LIN {X -0.020,Y -573.873,Z 1383.296,A 0.000,B 0.000,C 90.000,E1 89.312} C_DIS
LIN {X 0.144,Y -573.679,Z 1383.294,A 0.000,B 0.000,C 90.000,E1 88.854} C_DIS
LIN {X 0.149,Y -575.125,Z 1383.283,A 0.000,B 0.000,C 90.000,E1 86.963} C_DIS
LIN {X 0.133,Y -576.877,Z 1383.273,A 0.000,B 0.000,C 90.000,E1 85.065} C_DIS
LIN {X -0.055,Y -579.570,Z 1383.259,A 0.000,B 0.000,C 90.000,E1 82.648} C_DIS
LIN {X -0.182,Y -581.188,Z 1383.252,A 0.000,B 0.000,C 90.000,E1 81.310} C_DIS
LIN {X 0.204,Y -582.794,Z 1383.244,A 0.000,B 0.000,C 90.000,E1 79.926} C_DIS
LIN {X 0.003,Y -584.002,Z 1383.238,A 0.000,B 0.000,C 90.000,E1 78.870} C_DIS
LIN {X 0.074,Y -585.294,Z 1383.231,A 0.000,B 0.000,C 90.000,E1 77.521} C_DIS
LIN {X 0.163,Y -586.431,Z 1383.223,A 0.000,B 0.000,C 90.000,E1 76.172} C_DIS
LIN {X 0.161,Y -587.247,Z 1383.217,A 0.000,B 0.000,C 90.000,E1 75.102} C_DIS
LIN {X -0.143,Y -588.135,Z 1383.210,A 0.000,B 0.000,C 90.000,E1 73.795} C_DIS
LIN {X -0.346,Y -589.192,Z 1383.200,A 0.000,B 0.000,C 90.000,E1 71.945} C_DIS
LIN {X -0.162,Y -590.287,Z 1383.189,A 0.000,B 0.000,C 90.000,E1 70.061} C_DIS
LIN {X -0.073,Y -591.511,Z 1383.177,A 0.000,B 0.000,C 90.000,E1 67.922} C_DIS
LIN {X -0.049,Y -593.020,Z 1383.166,A 0.000,B 0.000,C 90.000,E1 65.793} C_DIS
LIN {X -0.080,Y -594.374,Z 1383.157,A 0.000,B 0.000,C 90.000,E1 64.204} C_DIS
LIN {X -0.086,Y -595.616,Z 1383.148,A 0.000,B 0.000,C 90.000,E1 62.615} C_DIS
LIN {X 0.354,Y -598.154,Z 1383.132,A 0.000,B 0.000,C 90.000,E1 59.665} C_DIS
LIN {X -0.139,Y -599.857,Z 1383.121,A 0.000,B 0.000,C 90.000,E1 57.867} C_DIS
LIN {X -0.197,Y -601.333,Z 1383.113,A 0.000,B 0.000,C 90.000,E1 56.294} C_DIS
LIN {X 0.366,Y -602.985,Z 1383.103,A 0.000,B 0.000,C 90.000,E1 54.402} C_DIS
LIN {X 0.223,Y -604.383,Z 1383.094,A 0.000,B 0.000,C 90.000,E1 52.844} C_DIS
LIN {X 0.156,Y -605.045,Z 1383.089,A 0.000,B 0.000,C 90.000,E1 52.065} C_DIS
LIN {X -0.005,Y -605.621,Z 1383.085,A 0.000,B 0.000,C 90.000,E1 51.295} C_DIS
LIN {X -0.206,Y -606.465,Z 1383.076,A 0.000,B 0.000,C 90.000,E1 49.747} C_DIS
LIN {X 0.188,Y -607.019,Z 1383.069,A 0.000,B 0.000,C 90.000,E1 48.405} C_DIS
LIN {X -0.066,Y -607.335,Z 1383.060,A 0.000,B 0.000,C 90.000,E1 46.863} C_DIS
LIN {X -0.150,Y -607.368,Z 1383.053,A 0.000,B 0.000,C 90.000,E1 45.567} C_DIS
LIN {X -0.039,Y -607.232,Z 1383.047,A 0.000,B 0.000,C 90.000,E1 44.514} C_DIS
LIN {X 0.065,Y -606.899,Z 1383.042,A 0.000,B 0.000,C 90.000,E1 43.461} C_DIS
LIN {X -0.256,Y -606.457,Z 1383.036,A 0.000,B 0.000,C 90.000,E1 42.447} C_DIS
LIN {X -0.066,Y -605.580,Z 1383.027,A 0.000,B 0.000,C 90.000,E1 40.862} C_DIS
LIN {X -0.152,Y -604.657,Z 1383.020,A 0.000,B 0.000,C 90.000,E1 39.564} C_DIS
LIN {X 0.157,Y -604.020,Z 1383.015,A 0.000,B 0.000,C 90.000,E1 38.749} C_DIS
LIN {X 0.122,Y -602.737,Z 1383.008,A 0.000,B 0.000,C 90.000,E1 37.443} C_DIS
LIN {X 0.061,Y -601.033,Z 1383.001,A 0.000,B 0.000,C 90.000,E1 36.137} C_DIS
LIN {X -0.040,Y -599.758,Z 1382.996,A 0.000,B 0.000,C 90.000,E1 35.358} C_DIS
LIN {X -0.002,Y -598.228,Z 1382.992,A 0.000,B 0.000,C 90.000,E1 34.565} C_DIS
LIN {X 0.101,Y -595.889,Z 1382.986,A 0.000,B 0.000,C 90.000,E1 33.499} C_DIS
LIN {X 0.221,Y -594.656,Z 1382.983,A 0.000,B 0.000,C 90.000,E1 32.959} C_DIS
LIN {X -0.175,Y -591.080,Z 1382.976,A 0.000,B 0.000,C 90.000,E1 31.671} C_DIS
LIN {X -0.086,Y -589.475,Z 1382.973,A 0.000,B 0.000,C 90.000,E1 31.131} C_DIS
LIN {X -0.127,Y -586.543,Z 1382.969,A 0.000,B 0.000,C 90.000,E1 30.335} C_DIS
LIN {X -0.197,Y -583.338,Z 1382.964,A 0.000,B 0.000,C 90.000,E1 29.539} C_DIS
LIN {X -0.169,Y -580.992,Z 1382.961,A 0.000,B 0.000,C 90.000,E1 28.999} C_DIS
LIN {X 0.203,Y -577.244,Z 1382.957,A 0.000,B 0.000,C 90.000,E1 28.153} C_DIS
LIN {X 0.183,Y -572.284,Z 1382.951,A 0.000,B 0.000,C 90.000,E1 27.206} C_DIS
LIN {X -0.143,Y -566.792,Z 1382.946,A 0.000,B 0.000,C 90.000,E1 26.283} C_DIS
LIN {X 0.003,Y -563.478,Z 1382.943,A 0.000,B 0.000,C 90.000,E1 25.720} C_DIS
LIN {X 0.127,Y -559.951,Z 1382.940,A 0.000,B 0.000,C 90.000,E1 25.155} C_DIS
LIN {X -0.278,Y -556.223,Z 1382.937,A 0.000,B 0.000,C 90.000,E1 24.643} C_DIS
LIN {X -0.203,Y -552.304,Z 1382.934,A 0.000,B 0.000,C 90.000,E1 24.079} C_DIS
LIN {X -0.040,Y -549.189,Z 1382.931,A 0.000,B 0.000,C 90.000,E1 23.643} C_DIS
LIN {X -0.017,Y -544.710,Z 1382.928,A 0.000,B 0.000,C 90.000,E1 23.078} C_DIS
LIN {X 0.218,Y -537.735,Z 1382.924,A 0.000,B 0.000,C 90.000,E1 22.206} C_DIS
LIN {X -0.045,Y -532.751,Z 1382.920,A 0.000,B 0.000,C 90.000,E1 21.663} C_DIS
LIN {X -0.050,Y -522.640,Z 1382.914,A 0.000,B 0.000,C 90.000,E1 20.556} C_DIS
LIN {X -0.068,Y -512.091,Z 1382.908,A 0.000,B 0.000,C 90.000,E1 19.450} C_DIS
LIN {X -0.052,Y -502.768,Z 1382.903,A 0.000,B 0.000,C 90.000,E1 18.489} C_DIS
LIN {X -0.109,Y -486.527,Z 1382.894,A 0.000,B 0.000,C 90.000,E1 16.858} C_DIS
LIN {X -0.241,Y -474.100,Z 1382.887,A 0.000,B 0.000,C 90.000,E1 15.607} C_DIS
LIN {X 0.115,Y -463.083,Z 1382.880,A 0.000,B 0.000,C 90.000,E1 14.426} C_DIS
LIN {X 0.044,Y -449.284,Z 1382.872,A 0.000,B 0.000,C 90.000,E1 13.008} C_DIS
LIN {X -0.001,Y -429.820,Z 1382.861,A 0.000,B 0.000,C 90.000,E1 10.894} C_DIS
LIN {X -0.006,Y -413.486,Z 1382.850,A 0.000,B 0.000,C 90.000,E1 8.973} C_DIS
LIN {X -0.053,Y -403.732,Z 1382.843,A 0.000,B 0.000,C 90.000,E1 7.814} C_DIS
LIN {X 0.113,Y -396.786,Z 1382.839,A 0.000,B 0.000,C 90.000,E1 6.947} C_DIS
LIN {X 0.110,Y -392.848,Z 1382.836,A 0.000,B 0.000,C 90.000,E1 6.429} C_DIS
LIN {X -0.156,Y -390.657,Z 1382.834,A 0.000,B 0.000,C 90.000,E1 6.087} C_DIS
LIN {X -0.193,Y -390.686,Z 1382.834,A 0.000,B 0.000,C 90.000,E1 6.087} C_DIS
LIN {X 0.157,Y -393.696,Z 1382.831,A 0.000,B 0.000,C 90.000,E1 5.625} C_DIS
LIN {X 0.158,Y -398.277,Z 1382.829,A 0.000,B 0.000,C 90.000,E1 5.220} C_DIS
LIN {X 0.115,Y -404.369,Z 1382.827,A 0.000,B 0.000,C 90.000,E1 4.759} C_DIS
LIN {X 0.005,Y -410.468,Z 1382.824,A 0.000,B 0.000,C 90.000,E1 4.245} C_DIS
LIN {X 0.154,Y -417.659,Z 1382.820,A 0.000,B 0.000,C 90.000,E1 3.498} C_DIS
LIN {X 0.153,Y -424.246,Z 1382.815,A 0.000,B 0.000,C 90.000,E1 2.694} C_DIS
LIN {X -0.070,Y -431.567,Z 1382.810,A 0.000,B 0.000,C 90.000,E1 1.718} C_DIS
LIN {X 0.135,Y -437.381,Z 1382.805,A 0.000,B 0.000,C 90.000,E1 0.859} C_DIS
LIN {X 0.000,Y -443.207,Z 1382.800,A 0.000,B 0.000,C 90.000,E1 360.000} C_DIS
LIN {X -0.007,Y -448.622,Z 1382.795,A 0.000,B 0.000,C 90.000,E1 359.141} C_DIS
LIN {X -0.072,Y -453.427,Z 1382.791,A 0.000,B 0.000,C 90.000,E1 358.339} C_DIS
LIN {X -0.079,Y -457.872,Z 1382.786,A 0.000,B 0.000,C 90.000,E1 357.535} C_DIS
LIN {X -0.037,Y -461.977,Z 1382.782,A 0.000,B 0.000,C 90.000,E1 356.731} C_DIS
LIN {X -0.089,Y -465.100,Z 1382.778,A 0.000,B 0.000,C 90.000,E1 356.102} C_DIS
LIN {X 0.021,Y -468.608,Z 1382.774,A 0.000,B 0.000,C 90.000,E1 355.298} C_DIS
LIN {X 0.211,Y -471.931,Z 1382.770,A 0.000,B 0.000,C 90.000,E1 354.489} C_DIS
LIN {X -0.082,Y -474.974,Z 1382.765,A 0.000,B 0.000,C 90.000,E1 353.742} C_DIS
LIN {X -0.176,Y -478.364,Z 1382.760,A 0.000,B 0.000,C 90.000,E1 352.818} C_DIS
LIN {X -0.079,Y -480.443,Z 1382.757,A 0.000,B 0.000,C 90.000,E1 352.186} C_DIS
LIN {X 0.100,Y -482.341,Z 1382.753,A 0.000,B 0.000,C 90.000,E1 351.546} C_DIS
LIN {X -0.042,Y -483.121,Z 1382.751,A 0.000,B 0.000,C 90.000,E1 351.254} C_DIS
LIN {X -0.255,Y -483.750,Z 1382.750,A 0.000,B 0.000,C 90.000,E1 350.971} C_DIS
LIN {X 0.085,Y -484.175,Z 1382.748,A 0.000,B 0.000,C 90.000,E1 350.622} C_DIS
LIN {X -0.048,Y -484.309,Z 1382.746,A 0.000,B 0.000,C 90.000,E1 350.330} C_DIS
LIN {X -0.179,Y -483.925,Z 1382.745,A 0.000,B 0.000,C 90.000,E1 350.038} C_DIS
LIN {X 0.037,Y -483.259,Z 1382.744,A 0.000,B 0.000,C 90.000,E1 349.859} C_DIS
LIN {X 0.166,Y -480.581,Z 1382.743,A 0.000,B 0.000,C 90.000,E1 349.690} C_DIS
LIN {X -0.004,Y -439.598,Z 1382.738,A 0.000,B 0.000,C 90.000,E1 348.757} C_DIS
LIN {X 0.119,Y -404.062,Z 1382.732,A 0.000,B 0.000,C 90.000,E1 347.757} C_DIS
LIN {X -0.141,Y -372.252,Z 1382.726,A 0.000,B 0.000,C 90.000,E1 346.756} C_DIS
LIN {X -0.087,Y -359.594,Z 1382.724,A 0.000,B 0.000,C 90.000,E1 346.284} C_DIS
LIN {X -0.114,Y -359.561,Z 1382.724,A 0.000,B 0.000,C 90.000,E1 346.284} C_DIS
LIN {X 0.021,Y -361.837,Z 1382.684,A 0.000,B 0.000,C 90.000,E1 339.082} C_DIS
LIN {X -0.077,Y -362.147,Z 1382.678,A 0.000,B 0.000,C 90.000,E1 337.975} C_DIS
LIN {X -0.130,Y -366.028,Z 1382.642,A 0.000,B 0.000,C 90.000,E1 331.641} C_DIS
LIN {X -0.029,Y -366.575,Z 1382.636,A 0.000,B 0.000,C 90.000,E1 330.511} C_DIS
LIN {X -0.136,Y -371.414,Z 1382.603,A 0.000,B 0.000,C 90.000,E1 324.609} C_DIS
LIN {X 0.155,Y -371.796,Z 1382.601,A 0.000,B 0.000,C 90.000,E1 324.196} C_DIS
LIN {X -0.057,Y -377.421,Z 1382.567,A 0.000,B 0.000,C 90.000,E1 318.000} C_DIS
LIN {X 0.224,Y -378.265,Z 1382.563,A 0.000,B 0.000,C 90.000,E1 317.229} C_DIS
LIN {X -0.034,Y -384.005,Z 1382.530,A 0.000,B 0.000,C 90.000,E1 311.472} C_DIS
LIN {X 0.014,Y -384.924,Z 1382.526,A 0.000,B 0.000,C 90.000,E1 310.744} C_DIS
LIN {X -0.065,Y -390.676,Z 1382.495,A 0.000,B 0.000,C 90.000,E1 305.025} C_DIS
LIN {X 0.002,Y -391.172,Z 1382.493,A 0.000,B 0.000,C 90.000,E1 304.659} C_DIS
LIN {X -0.156,Y -394.014,Z 1382.473,A 0.000,B 0.000,C 90.000,E1 301.131} C_DIS
LIN {X 0.130,Y -396.888,Z 1382.459,A 0.000,B 0.000,C 90.000,E1 298.615} C_DIS
LIN {X -0.093,Y -397.488,Z 1382.453,A 0.000,B 0.000,C 90.000,E1 297.590} C_DIS
LIN {X 0.141,Y -401.629,Z 1382.426,A 0.000,B 0.000,C 90.000,E1 292.642} C_DIS
LIN {X -0.109,Y -404.701,Z 1382.395,A 0.000,B 0.000,C 90.000,E1 287.094} C_DIS
LIN {X 0.075,Y -405.163,Z 1382.376,A 0.000,B 0.000,C 90.000,E1 283.592} C_DIS
LIN {X -0.116,Y -406.127,Z 1382.364,A 0.000,B 0.000,C 90.000,E1 281.535} C_DIS
LIN {X -0.084,Y -405.826,Z 1382.358,A 0.000,B 0.000,C 90.000,E1 280.489} C_DIS
LIN {X -0.024,Y -405.689,Z 1382.333,A 0.000,B 0.000,C 90.000,E1 275.967} C_DIS
LIN {X 0.014,Y -403.467,Z 1382.304,A 0.000,B 0.000,C 90.000,E1 270.745} C_DIS
LIN {X -0.019,Y -403.254,Z 1382.302,A 0.000,B 0.000,C 90.000,E1 270.401} C_DIS
LIN {X 0.160,Y -398.876,Z 1382.271,A 0.000,B 0.000,C 90.000,E1 264.780} C_DIS
LIN {X 0.058,Y -393.350,Z 1382.244,A 0.000,B 0.000,C 90.000,E1 259.859} C_DIS
LIN {X -0.020,Y -392.780,Z 1382.240,A 0.000,B 0.000,C 90.000,E1 259.162} C_DIS
LIN {X 0.058,Y -386.327,Z 1382.214,A 0.000,B 0.000,C 90.000,E1 254.519} C_DIS
LIN {X 0.020,Y -385.221,Z 1382.208,A 0.000,B 0.000,C 90.000,E1 253.449} C_DIS
LIN {X 0.060,Y -384.022,Z 1382.204,A 0.000,B 0.000,C 90.000,E1 252.725} C_DIS
LIN {X -0.111,Y -377.452,Z 1382.180,A 0.000,B 0.000,C 90.000,E1 248.411} C_DIS
LIN {X -0.018,Y -376.179,Z 1382.174,A 0.000,B 0.000,C 90.000,E1 247.305} C_DIS
LIN {X -0.030,Y -368.350,Z 1382.147,A 0.000,B 0.000,C 90.000,E1 242.538} C_DIS
LIN {X 0.014,Y -366.486,Z 1382.139,A 0.000,B 0.000,C 90.000,E1 241.051} C_DIS
LIN {X 0.098,Y -365.950,Z 1382.137,A 0.000,B 0.000,C 90.000,E1 240.667} C_DIS
LIN {X -0.012,Y -359.125,Z 1382.114,A 0.000,B 0.000,C 90.000,E1 236.580} C_DIS
LIN {X -0.017,Y -356.266,Z 1382.102,A 0.000,B 0.000,C 90.000,E1 234.322} C_DIS
LIN {X 0.204,Y -355.749,Z 1382.100,A 0.000,B 0.000,C 90.000,E1 233.909} C_DIS
LIN {X 0.006,Y -348.729,Z 1382.074,A 0.000,B 0.000,C 90.000,E1 229.380} C_DIS
LIN {X 0.080,Y -346.133,Z 1382.062,A 0.000,B 0.000,C 90.000,E1 227.067} C_DIS
LIN {X 0.207,Y -344.385,Z 1382.055,A 0.000,B 0.000,C 90.000,E1 225.891} C_DIS
LIN {X -0.130,Y -338.157,Z 1382.027,A 0.000,B 0.000,C 90.000,E1 220.906} C_DIS
LIN {X -0.002,Y -336.778,Z 1382.019,A 0.000,B 0.000,C 90.000,E1 219.322} C_DIS
LIN {X -0.107,Y -330.820,Z 1381.988,A 0.000,B 0.000,C 90.000,E1 213.833} C_DIS
LIN {X -0.157,Y -329.265,Z 1381.975,A 0.000,B 0.000,C 90.000,E1 211.465} C_DIS
LIN {X -0.025,Y -324.644,Z 1381.942,A 0.000,B 0.000,C 90.000,E1 205.463} C_DIS
LIN {X -0.130,Y -323.816,Z 1381.928,A 0.000,B 0.000,C 90.000,E1 203.078} C_DIS
LIN {X 0.102,Y -321.071,Z 1381.888,A 0.000,B 0.000,C 90.000,E1 195.843} C_DIS
LIN {X 0.085,Y -321.097,Z 1381.888,A 0.000,B 0.000,C 90.000,E1 195.843} C_DIS
LIN {X -0.157,Y -345.481,Z 1381.882,A 0.000,B 0.000,C 90.000,E1 194.773} C_DIS
LIN {X 0.193,Y -372.735,Z 1381.876,A 0.000,B 0.000,C 90.000,E1 193.647} C_DIS
LIN {X -0.083,Y -401.975,Z 1381.871,A 0.000,B 0.000,C 90.000,E1 192.703} C_DIS
LIN {X 0.166,Y -434.993,Z 1381.865,A 0.000,B 0.000,C 90.000,E1 191.715} C_DIS
LIN {X -0.147,Y -438.036,Z 1381.865,A 0.000,B 0.000,C 90.000,E1 191.658} C_DIS
LIN {X -0.077,Y -439.089,Z 1381.864,A 0.000,B 0.000,C 90.000,E1 191.535} C_DIS
LIN {X -0.202,Y -440.356,Z 1381.862,A 0.000,B 0.000,C 90.000,E1 191.243} C_DIS
LIN {X -0.054,Y -440.972,Z 1381.860,A 0.000,B 0.000,C 90.000,E1 190.894} C_DIS
LIN {X 0.100,Y -441.221,Z 1381.859,A 0.000,B 0.000,C 90.000,E1 190.546} C_DIS
LIN {X -0.019,Y -441.141,Z 1381.855,A 0.000,B 0.000,C 90.000,E1 189.905} C_DIS
LIN {X -0.012,Y -440.794,Z 1381.844,A 0.000,B 0.000,C 90.000,E1 187.936} C_DIS
LIN {X -0.171,Y -440.447,Z 1381.835,A 0.000,B 0.000,C 90.000,E1 186.315} C_DIS
LIN {X -0.100,Y -440.032,Z 1381.828,A 0.000,B 0.000,C 90.000,E1 184.992} C_DIS
LIN {X 0.152,Y -439.714,Z 1381.824,A 0.000,B 0.000,C 90.000,E1 184.302} C_DIS
LIN {X -0.038,Y -439.218,Z 1381.820,A 0.000,B 0.000,C 90.000,E1 183.669} C_DIS
LIN {X -0.126,Y -438.097,Z 1381.815,A 0.000,B 0.000,C 90.000,E1 182.694} C_DIS
LIN {X -0.125,Y -436.311,Z 1381.808,A 0.000,B 0.000,C 90.000,E1 181.375} C_DIS
LIN {X 0.076,Y -435.150,Z 1381.804,A 0.000,B 0.000,C 90.000,E1 180.688} C_DIS
LIN {X -0.165,Y -433.828,Z 1381.800,A 0.000,B 0.000,C 90.000,E1 180.057} C_DIS
LIN {X 0.019,Y -432.334,Z 1381.797,A 0.000,B 0.000,C 90.000,E1 179.370} C_DIS
LIN {X 0.189,Y -430.598,Z 1381.793,A 0.000,B 0.000,C 90.000,E1 178.682} C_DIS
LIN {X -0.001,Y -427.494,Z 1381.787,A 0.000,B 0.000,C 90.000,E1 177.707} C_DIS
LIN {X 0.153,Y -424.395,Z 1381.783,A 0.000,B 0.000,C 90.000,E1 176.849} C_DIS
LIN {X -0.132,Y -420.678,Z 1381.778,A 0.000,B 0.000,C 90.000,E1 176.045} C_DIS
LIN {X 0.000,Y -416.285,Z 1381.773,A 0.000,B 0.000,C 90.000,E1 175.179} C_DIS
LIN {X 0.050,Y -410.147,Z 1381.768,A 0.000,B 0.000,C 90.000,E1 174.147} C_DIS
LIN {X 0.140,Y -398.792,Z 1381.758,A 0.000,B 0.000,C 90.000,E1 172.413} C_DIS
LIN {X -0.071,Y -386.807,Z 1381.747,A 0.000,B 0.000,C 90.000,E1 170.500} C_DIS
LIN {X 0.012,Y -379.002,Z 1381.739,A 0.000,B 0.000,C 90.000,E1 169.050} C_DIS
LIN {X -0.094,Y -376.326,Z 1381.736,A 0.000,B 0.000,C 90.000,E1 168.522} C_DIS
LIN {X -0.041,Y -374.329,Z 1381.733,A 0.000,B 0.000,C 90.000,E1 167.993} C_DIS
LIN {X 0.172,Y -373.011,Z 1381.731,A 0.000,B 0.000,C 90.000,E1 167.521} C_DIS
LIN {X 0.135,Y -373.003,Z 1381.731,A 0.000,B 0.000,C 90.000,E1 167.521} C_DIS
LIN {X 0.176,Y -373.367,Z 1381.729,A 0.000,B 0.000,C 90.000,E1 167.229} C_DIS
LIN {X -0.114,Y -373.475,Z 1381.728,A 0.000,B 0.000,C 90.000,E1 166.992} C_DIS
LIN {X -0.151,Y -373.500,Z 1381.728,A 0.000,B 0.000,C 90.000,E1 166.992} C_DIS
LIN {X 0.019,Y -375.985,Z 1381.725,A 0.000,B 0.000,C 90.000,E1 166.520} C_DIS
LIN {X 0.092,Y -380.278,Z 1381.722,A 0.000,B 0.000,C 90.000,E1 165.936} C_DIS
LIN {X -0.059,Y -387.164,Z 1381.718,A 0.000,B 0.000,C 90.000,E1 165.172} C_DIS
LIN {X 0.124,Y -399.186,Z 1381.711,A 0.000,B 0.000,C 90.000,E1 163.921} C_DIS
LIN {X 0.126,Y -416.360,Z 1381.702,A 0.000,B 0.000,C 90.000,E1 162.362} C_DIS
LIN {X -0.141,Y -440.127,Z 1381.692,A 0.000,B 0.000,C 90.000,E1 160.477} C_DIS
LIN {X -0.186,Y -452.554,Z 1381.686,A 0.000,B 0.000,C 90.000,E1 159.518} C_DIS
LIN {X -0.109,Y -461.794,Z 1381.682,A 0.000,B 0.000,C 90.000,E1 158.773} C_DIS
LIN {X -0.214,Y -467.844,Z 1381.679,A 0.000,B 0.000,C 90.000,E1 158.284} C_DIS
LIN {X 0.106,Y -475.197,Z 1381.676,A 0.000,B 0.000,C 90.000,E1 157.614} C_DIS
LIN {X -0.085,Y -483.917,Z 1381.671,A 0.000,B 0.000,C 90.000,E1 156.847} C_DIS
LIN {X 0.146,Y -493.943,Z 1381.666,A 0.000,B 0.000,C 90.000,E1 155.869} C_DIS
LIN {X -0.013,Y -502.075,Z 1381.661,A 0.000,B 0.000,C 90.000,E1 155.049} C_DIS
LIN {X 0.106,Y -505.969,Z 1381.659,A 0.000,B 0.000,C 90.000,E1 154.613} C_DIS
LIN {X -0.218,Y -513.623,Z 1381.654,A 0.000,B 0.000,C 90.000,E1 153.768} C_DIS
LIN {X 0.072,Y -519.639,Z 1381.650,A 0.000,B 0.000,C 90.000,E1 152.999} C_DIS
LIN {X 0.037,Y -523.026,Z 1381.648,A 0.000,B 0.000,C 90.000,E1 152.564} C_DIS
LIN {X 0.105,Y -527.199,Z 1381.644,A 0.000,B 0.000,C 90.000,E1 151.975} C_DIS
LIN {X 0.206,Y -530.879,Z 1381.641,A 0.000,B 0.000,C 90.000,E1 151.385} C_DIS
LIN {X -0.129,Y -534.105,Z 1381.638,A 0.000,B 0.000,C 90.000,E1 150.845} C_DIS
LIN {X 0.026,Y -536.888,Z 1381.635,A 0.000,B 0.000,C 90.000,E1 150.255} C_DIS
LIN {X -0.073,Y -540.427,Z 1381.630,A 0.000,B 0.000,C 90.000,E1 149.410} C_DIS
LIN {X 0.121,Y -542.498,Z 1381.627,A 0.000,B 0.000,C 90.000,E1 148.820} C_DIS
LIN {X 0.149,Y -544.391,Z 1381.624,A 0.000,B 0.000,C 90.000,E1 148.250} C_DIS
LIN {X 0.109,Y -546.661,Z 1381.619,A 0.000,B 0.000,C 90.000,E1 147.406} C_DIS
LIN {X 0.180,Y -548.004,Z 1381.616,A 0.000,B 0.000,C 90.000,E1 146.834} C_DIS
LIN {X 0.011,Y -549.716,Z 1381.611,A 0.000,B 0.000,C 90.000,E1 146.008} C_DIS
LIN {X -0.196,Y -550.735,Z 1381.608,A 0.000,B 0.000,C 90.000,E1 145.468} C_DIS
LIN {X 0.037,Y -552.308,Z 1381.602,A 0.000,B 0.000,C 90.000,E1 144.322} C_DIS
LIN {X -0.160,Y -552.962,Z 1381.599,A 0.000,B 0.000,C 90.000,E1 143.783} C_DIS
LIN {X 0.108,Y -553.981,Z 1381.593,A 0.000,B 0.000,C 90.000,E1 142.637} C_DIS
LIN {X 0.095,Y -555.227,Z 1381.583,A 0.000,B 0.000,C 90.000,E1 140.964} C_DIS
LIN {X -0.039,Y -556.124,Z 1381.576,A 0.000,B 0.000,C 90.000,E1 139.585} C_DIS
LIN {X -0.074,Y -556.991,Z 1381.566,A 0.000,B 0.000,C 90.000,E1 137.919} C_DIS
LIN {X -0.175,Y -557.566,Z 1381.558,A 0.000,B 0.000,C 90.000,E1 136.539} C_DIS
LIN {X 0.163,Y -558.196,Z 1381.549,A 0.000,B 0.000,C 90.000,E1 134.838} C_DIS
LIN {X 0.061,Y -558.713,Z 1381.542,A 0.000,B 0.000,C 90.000,E1 133.461} C_DIS
LIN {X -0.011,Y -559.084,Z 1381.534,A 0.000,B 0.000,C 90.000,E1 132.081} C_DIS
LIN {X -0.070,Y -559.395,Z 1381.526,A 0.000,B 0.000,C 90.000,E1 130.701} C_DIS
LIN {X -0.123,Y -560.425,Z 1381.511,A 0.000,B 0.000,C 90.000,E1 127.935} C_DIS
LIN {X 0.065,Y -561.015,Z 1381.508,A 0.000,B 0.000,C 90.000,E1 127.363} C_DIS
LIN {X 0.160,Y -561.930,Z 1381.506,A 0.000,B 0.000,C 90.000,E1 127.076} C_DIS
LIN {X 0.173,Y -562.481,Z 1381.505,A 0.000,B 0.000,C 90.000,E1 126.790} C_DIS
LIN {X 0.131,Y -562.526,Z 1381.505,A 0.000,B 0.000,C 90.000,E1 126.790} C_DIS
LIN {X 0.028,Y -563.550,Z 1381.504,A 0.000,B 0.000,C 90.000,E1 126.710} C_DIS
LIN {X 0.110,Y -569.997,Z 1381.503,A 0.000,B 0.000,C 90.000,E1 126.457} C_DIS
LIN {X -0.098,Y -579.785,Z 1381.501,A 0.000,B 0.000,C 90.000,E1 126.217} C_DIS
LIN {X 0.251,Y -582.362,Z 1381.501,A 0.000,B 0.000,C 90.000,E1 126.091} C_DIS
LIN {X -0.258,Y -588.367,Z 1381.499,A 0.000,B 0.000,C 90.000,E1 125.884} C_DIS
LIN {X -0.073,Y -591.151,Z 1381.499,A 0.000,B 0.000,C 90.000,E1 125.724} C_DIS
LIN {X 0.346,Y -594.060,Z 1381.498,A 0.000,B 0.000,C 90.000,E1 125.518} C_DIS
LIN {X -0.120,Y -599.752,Z 1381.495,A 0.000,B 0.000,C 90.000,E1 125.185} C_DIS
LIN {X -0.077,Y -604.019,Z 1381.494,A 0.000,B 0.000,C 90.000,E1 124.865} C_DIS
LIN {X 0.058,Y -609.454,Z 1381.491,A 0.000,B 0.000,C 90.000,E1 124.405} C_DIS
LIN {X -0.097,Y -617.243,Z 1381.487,A 0.000,B 0.000,C 90.000,E1 123.706} C_DIS
LIN {X -0.097,Y -622.157,Z 1381.484,A 0.000,B 0.000,C 90.000,E1 123.214} C_DIS
LIN {X 0.227,Y -627.868,Z 1381.481,A 0.000,B 0.000,C 90.000,E1 122.546} C_DIS
LIN {X -0.297,Y -631.133,Z 1381.479,A 0.000,B 0.000,C 90.000,E1 122.212} C_DIS
LIN {X -0.417,Y -637.998,Z 1381.474,A 0.000,B 0.000,C 90.000,E1 121.337} C_DIS
LIN {X 0.034,Y -642.421,Z 1381.470,A 0.000,B 0.000,C 90.000,E1 120.669} C_DIS
LIN {X -0.035,Y -646.297,Z 1381.467,A 0.000,B 0.000,C 90.000,E1 120.050} C_DIS
LIN {X 0.166,Y -649.593,Z 1381.464,A 0.000,B 0.000,C 90.000,E1 119.411} C_DIS
LIN {X -0.171,Y -652.380,Z 1381.460,A 0.000,B 0.000,C 90.000,E1 118.821} C_DIS
LIN {X 0.033,Y -654.061,Z 1381.457,A 0.000,B 0.000,C 90.000,E1 118.309} C_DIS
LIN {X -0.327,Y -655.509,Z 1381.455,A 0.000,B 0.000,C 90.000,E1 117.847} C_DIS
LIN {X 0.020,Y -656.508,Z 1381.450,A 0.000,B 0.000,C 90.000,E1 117.078} C_DIS
LIN {X 0.139,Y -656.689,Z 1381.449,A 0.000,B 0.000,C 90.000,E1 116.821} C_DIS
LIN {X -0.090,Y -656.521,Z 1381.445,A 0.000,B 0.000,C 90.000,E1 116.104} C_DIS
LIN {X 0.148,Y -656.182,Z 1381.442,A 0.000,B 0.000,C 90.000,E1 115.591} C_DIS
LIN {X 0.265,Y -655.954,Z 1381.441,A 0.000,B 0.000,C 90.000,E1 115.335} C_DIS
LIN {X -0.375,Y -655.110,Z 1381.438,A 0.000,B 0.000,C 90.000,E1 114.899} C_DIS
LIN {X -0.261,Y -654.591,Z 1381.437,A 0.000,B 0.000,C 90.000,E1 114.643} C_DIS
LIN {X 0.012,Y -651.678,Z 1381.433,A 0.000,B 0.000,C 90.000,E1 114.003} C_DIS
LIN {X -0.056,Y -647.230,Z 1381.431,A 0.000,B 0.000,C 90.000,E1 113.515} C_DIS
LIN {X -0.011,Y -645.868,Z 1381.430,A 0.000,B 0.000,C 90.000,E1 113.387} C_DIS
LIN {X -0.021,Y -641.544,Z 1381.429,A 0.000,B 0.000,C 90.000,E1 113.153} C_DIS
LIN {X 0.184,Y -636.673,Z 1381.427,A 0.000,B 0.000,C 90.000,E1 112.898} C_DIS
LIN {X 0.131,Y -631.213,Z 1381.426,A 0.000,B 0.000,C 90.000,E1 112.717} C_DIS
LIN {X 0.064,Y -617.234,Z 1381.424,A 0.000,B 0.000,C 90.000,E1 112.333} C_DIS
LIN {X 0.001,Y -617.209,Z 1381.424,A 0.000,B 0.000,C 90.000,E1 112.333} C_DIS
LIN {X -0.151,Y -623.404,Z 1381.421,A 0.000,B 0.000,C 90.000,E1 111.716} C_DIS
LIN {X 0.198,Y -627.890,Z 1381.418,A 0.000,B 0.000,C 90.000,E1 111.227} C_DIS
LIN {X 0.039,Y -631.423,Z 1381.416,A 0.000,B 0.000,C 90.000,E1 110.865} C_DIS
LIN {X -0.133,Y -636.709,Z 1381.412,A 0.000,B 0.000,C 90.000,E1 110.248} C_DIS
LIN {X -0.238,Y -641.308,Z 1381.409,A 0.000,B 0.000,C 90.000,E1 109.631} C_DIS
LIN {X 0.083,Y -646.030,Z 1381.405,A 0.000,B 0.000,C 90.000,E1 108.852} C_DIS
LIN {X -0.123,Y -650.949,Z 1381.400,A 0.000,B 0.000,C 90.000,E1 108.000} C_DIS
LIN {X 0.339,Y -655.241,Z 1381.395,A 0.000,B 0.000,C 90.000,E1 107.094} C_DIS
LIN {X -0.012,Y -658.153,Z 1381.391,A 0.000,B 0.000,C 90.000,E1 106.386} C_DIS
LIN {X -0.046,Y -659.626,Z 1381.388,A 0.000,B 0.000,C 90.000,E1 105.898} C_DIS
LIN {X -0.353,Y -661.325,Z 1381.384,A 0.000,B 0.000,C 90.000,E1 105.190} C_DIS
LIN {X 0.002,Y -662.557,Z 1381.380,A 0.000,B 0.000,C 90.000,E1 104.426} C_DIS
LIN {X -0.021,Y -663.206,Z 1381.377,A 0.000,B 0.000,C 90.000,E1 103.939} C_DIS
LIN {X -0.203,Y -663.683,Z 1381.375,A 0.000,B 0.000,C 90.000,E1 103.467} C_DIS
LIN {X 0.028,Y -663.975,Z 1381.371,A 0.000,B 0.000,C 90.000,E1 102.715} C_DIS
LIN {X -0.147,Y -663.951,Z 1381.368,A 0.000,B 0.000,C 90.000,E1 102.243} C_DIS
LIN {X -0.324,Y -663.729,Z 1381.365,A 0.000,B 0.000,C 90.000,E1 101.771} C_DIS
LIN {X 0.053,Y -662.928,Z 1381.361,A 0.000,B 0.000,C 90.000,E1 101.007} C_DIS
LIN {X -0.260,Y -662.226,Z 1381.359,A 0.000,B 0.000,C 90.000,E1 100.546} C_DIS
LIN {X 0.195,Y -661.236,Z 1381.356,A 0.000,B 0.000,C 90.000,E1 100.018} C_DIS
LIN {X -0.122,Y -660.068,Z 1381.353,A 0.000,B 0.000,C 90.000,E1 99.557} C_DIS
LIN {X 0.098,Y -657.885,Z 1381.349,A 0.000,B 0.000,C 90.000,E1 98.803} C_DIS
LIN {X -0.232,Y -656.211,Z 1381.346,A 0.000,B 0.000,C 90.000,E1 98.341} C_DIS
LIN {X 0.168,Y -654.322,Z 1381.344,A 0.000,B 0.000,C 90.000,E1 97.814} C_DIS
LIN {X -0.184,Y -652.193,Z 1381.341,A 0.000,B 0.000,C 90.000,E1 97.352} C_DIS
LIN {X -0.126,Y -648.582,Z 1381.337,A 0.000,B 0.000,C 90.000,E1 96.606} C_DIS
LIN {X 0.131,Y -645.841,Z 1381.334,A 0.000,B 0.000,C 90.000,E1 96.087} C_DIS
LIN {X 0.246,Y -642.240,Z 1381.330,A 0.000,B 0.000,C 90.000,E1 95.454} C_DIS
LIN {X 0.134,Y -636.874,Z 1381.326,A 0.000,B 0.000,C 90.000,E1 94.588} C_DIS
LIN {X 0.168,Y -632.492,Z 1381.322,A 0.000,B 0.000,C 90.000,E1 93.955} C_DIS
LIN {X -0.261,Y -628.532,Z 1381.319,A 0.000,B 0.000,C 90.000,E1 93.498} C_DIS
LIN {X -0.294,Y -622.636,Z 1381.316,A 0.000,B 0.000,C 90.000,E1 92.865} C_DIS
LIN {X -0.153,Y -616.126,Z 1381.312,A 0.000,B 0.000,C 90.000,E1 92.236} C_DIS
LIN {X 0.268,Y -609.623,Z 1381.309,A 0.000,B 0.000,C 90.000,E1 91.604} C_DIS
LIN {X 0.112,Y -604.109,Z 1381.307,A 0.000,B 0.000,C 90.000,E1 91.146} C_DIS
LIN {X 0.183,Y -599.489,Z 1381.305,A 0.000,B 0.000,C 90.000,E1 90.802} C_DIS
LIN {X -0.181,Y -596.399,Z 1381.303,A 0.000,B 0.000,C 90.000,E1 90.630} C_DIS
LIN {X -0.172,Y -591.380,Z 1381.302,A 0.000,B 0.000,C 90.000,E1 90.344} C_DIS
LIN {X -0.235,Y -587.734,Z 1381.301,A 0.000,B 0.000,C 90.000,E1 90.172} C_DIS
LIN {X -0.225,Y -582.641,Z 1381.300,A 0.000,B 0.000,C 90.000,E1 89.943} C_DIS
LIN {X -0.128,Y -578.416,Z 1381.298,A 0.000,B 0.000,C 90.000,E1 89.714} C_DIS
LIN {X 0.178,Y -577.051,Z 1381.298,A 0.000,B 0.000,C 90.000,E1 89.599} C_DIS
LIN {X -0.083,Y -574.787,Z 1381.297,A 0.000,B 0.000,C 90.000,E1 89.427} C_DIS
LIN {X -0.097,Y -573.959,Z 1381.296,A 0.000,B 0.000,C 90.000,E1 89.255} C_DIS
LIN {X 0.026,Y -573.666,Z 1381.294,A 0.000,B 0.000,C 90.000,E1 88.854} C_DIS
LIN {X 0.209,Y -575.282,Z 1381.282,A 0.000,B 0.000,C 90.000,E1 86.674} C_DIS
LIN {X 0.252,Y -576.278,Z 1381.276,A 0.000,B 0.000,C 90.000,E1 85.584} C_DIS
LIN {X 0.271,Y -578.238,Z 1381.265,A 0.000,B 0.000,C 90.000,E1 83.685} C_DIS
LIN {X 0.259,Y -580.168,Z 1381.256,A 0.000,B 0.000,C 90.000,E1 82.064} C_DIS
LIN {X 0.291,Y -582.106,Z 1381.247,A 0.000,B 0.000,C 90.000,E1 80.443} C_DIS
LIN {X 0.214,Y -583.660,Z 1381.240,A 0.000,B 0.000,C 90.000,E1 79.106} C_DIS
LIN {X 0.276,Y -585.003,Z 1381.232,A 0.000,B 0.000,C 90.000,E1 77.757} C_DIS
LIN {X 0.037,Y -586.399,Z 1381.223,A 0.000,B 0.000,C 90.000,E1 76.172} C_DIS
LIN {X 0.282,Y -587.398,Z 1381.216,A 0.000,B 0.000,C 90.000,E1 74.810} C_DIS
LIN {X 0.294,Y -588.103,Z 1381.210,A 0.000,B 0.000,C 90.000,E1 73.740} C_DIS
LIN {X 0.084,Y -589.161,Z 1381.199,A 0.000,B 0.000,C 90.000,E1 71.891} C_DIS
LIN {X -0.292,Y -590.254,Z 1381.189,A 0.000,B 0.000,C 90.000,E1 70.061} C_DIS
LIN {X -0.312,Y -591.636,Z 1381.176,A 0.000,B 0.000,C 90.000,E1 67.667} C_DIS
LIN {X -0.182,Y -592.994,Z 1381.166,A 0.000,B 0.000,C 90.000,E1 65.793} C_DIS
LIN {X -0.213,Y -594.354,Z 1381.157,A 0.000,B 0.000,C 90.000,E1 64.204} C_DIS
LIN {X -0.220,Y -595.558,Z 1381.148,A 0.000,B 0.000,C 90.000,E1 62.615} C_DIS
LIN {X 0.003,Y -597.890,Z 1381.133,A 0.000,B 0.000,C 90.000,E1 59.950} C_DIS
LIN {X -0.190,Y -599.608,Z 1381.123,A 0.000,B 0.000,C 90.000,E1 58.122} C_DIS
LIN {X -0.335,Y -601.344,Z 1381.113,A 0.000,B 0.000,C 90.000,E1 56.294} C_DIS
LIN {X -0.359,Y -603.207,Z 1381.101,A 0.000,B 0.000,C 90.000,E1 54.196} C_DIS
LIN {X -0.244,Y -604.851,Z 1381.091,A 0.000,B 0.000,C 90.000,E1 52.351} C_DIS
LIN {X -0.144,Y -605.627,Z 1381.085,A 0.000,B 0.000,C 90.000,E1 51.295} C_DIS
LIN {X 0.117,Y -606.435,Z 1381.076,A 0.000,B 0.000,C 90.000,E1 49.703} C_DIS
LIN {X 0.047,Y -606.979,Z 1381.069,A 0.000,B 0.000,C 90.000,E1 48.405} C_DIS
LIN {X 0.208,Y -607.334,Z 1381.060,A 0.000,B 0.000,C 90.000,E1 46.824} C_DIS
LIN {X -0.046,Y -607.374,Z 1381.052,A 0.000,B 0.000,C 90.000,E1 45.283} C_DIS
LIN {X -0.368,Y -607.180,Z 1381.046,A 0.000,B 0.000,C 90.000,E1 44.271} C_DIS
LIN {X 0.177,Y -606.801,Z 1381.040,A 0.000,B 0.000,C 90.000,E1 43.176} C_DIS
LIN {X -0.140,Y -606.321,Z 1381.034,A 0.000,B 0.000,C 90.000,E1 42.162} C_DIS
LIN {X 0.190,Y -605.598,Z 1381.027,A 0.000,B 0.000,C 90.000,E1 40.825} C_DIS
LIN {X -0.291,Y -604.682,Z 1381.020,A 0.000,B 0.000,C 90.000,E1 39.564} C_DIS
LIN {X 0.018,Y -604.057,Z 1381.015,A 0.000,B 0.000,C 90.000,E1 38.749} C_DIS
LIN {X -0.271,Y -603.060,Z 1381.010,A 0.000,B 0.000,C 90.000,E1 37.729} C_DIS
LIN {X -0.094,Y -601.791,Z 1381.004,A 0.000,B 0.000,C 90.000,E1 36.664} C_DIS
LIN {X -0.181,Y -600.714,Z 1380.999,A 0.000,B 0.000,C 90.000,E1 35.884} C_DIS
LIN {X -0.277,Y -599.385,Z 1380.995,A 0.000,B 0.000,C 90.000,E1 35.105} C_DIS
LIN {X 0.102,Y -597.791,Z 1380.990,A 0.000,B 0.000,C 90.000,E1 34.278} C_DIS
LIN {X 0.089,Y -594.765,Z 1380.983,A 0.000,B 0.000,C 90.000,E1 32.959} C_DIS
LIN {X -0.303,Y -591.160,Z 1380.976,A 0.000,B 0.000,C 90.000,E1 31.671} C_DIS
LIN {X -0.214,Y -589.577,Z 1380.973,A 0.000,B 0.000,C 90.000,E1 31.131} C_DIS
LIN {X -0.253,Y -586.663,Z 1380.968,A 0.000,B 0.000,C 90.000,E1 30.335} C_DIS
LIN {X -0.321,Y -583.442,Z 1380.964,A 0.000,B 0.000,C 90.000,E1 29.539} C_DIS
LIN {X 0.085,Y -579.873,Z 1380.959,A 0.000,B 0.000,C 90.000,E1 28.693} C_DIS
LIN {X 0.009,Y -576.642,Z 1380.956,A 0.000,B 0.000,C 90.000,E1 28.025} C_DIS
LIN {X -0.015,Y -571.687,Z 1380.950,A 0.000,B 0.000,C 90.000,E1 27.078} C_DIS
LIN {X 0.071,Y -565.331,Z 1380.944,A 0.000,B 0.000,C 90.000,E1 25.976} C_DIS
LIN {X 0.112,Y -560.992,Z 1380.941,A 0.000,B 0.000,C 90.000,E1 25.283} C_DIS
LIN {X 0.117,Y -556.337,Z 1380.937,A 0.000,B 0.000,C 90.000,E1 24.591} C_DIS
LIN {X 0.080,Y -551.401,Z 1380.933,A 0.000,B 0.000,C 90.000,E1 23.898} C_DIS
LIN {X 0.000,Y -546.034,Z 1380.929,A 0.000,B 0.000,C 90.000,E1 23.206} C_DIS
LIN {X 0.098,Y -537.822,Z 1380.923,A 0.000,B 0.000,C 90.000,E1 22.206} C_DIS
LIN {X -0.162,Y -532.883,Z 1380.920,A 0.000,B 0.000,C 90.000,E1 21.663} C_DIS
LIN {X -0.158,Y -522.525,Z 1380.914,A 0.000,B 0.000,C 90.000,E1 20.536} C_DIS
LIN {X 0.019,Y -511.863,Z 1380.908,A 0.000,B 0.000,C 90.000,E1 19.396} C_DIS
LIN {X 0.111,Y -503.666,Z 1380.903,A 0.000,B 0.000,C 90.000,E1 18.544} C_DIS
LIN {X 0.070,Y -491.550,Z 1380.896,A 0.000,B 0.000,C 90.000,E1 17.330} C_DIS
LIN {X -0.127,Y -479.031,Z 1380.889,A 0.000,B 0.000,C 90.000,E1 16.079} C_DIS
LIN {X -0.152,Y -465.028,Z 1380.881,A 0.000,B 0.000,C 90.000,E1 14.647} C_DIS
LIN {X 0.125,Y -455.048,Z 1380.876,A 0.000,B 0.000,C 90.000,E1 13.592} C_DIS
LIN {X 0.231,Y -438.499,Z 1380.866,A 0.000,B 0.000,C 90.000,E1 11.827} C_DIS
LIN {X -0.073,Y -417.757,Z 1380.853,A 0.000,B 0.000,C 90.000,E1 9.500} C_DIS
LIN {X -0.085,Y -408.020,Z 1380.846,A 0.000,B 0.000,C 90.000,E1 8.341} C_DIS
LIN {X -0.159,Y -399.550,Z 1380.841,A 0.000,B 0.000,C 90.000,E1 7.352} C_DIS
LIN {X 0.053,Y -394.836,Z 1380.837,A 0.000,B 0.000,C 90.000,E1 6.720} C_DIS
LIN {X 0.024,Y -392.300,Z 1380.835,A 0.000,B 0.000,C 90.000,E1 6.372} C_DIS
LIN {X -0.120,Y -390.927,Z 1380.834,A 0.000,B 0.000,C 90.000,E1 6.144} C_DIS
LIN {X -0.158,Y -390.915,Z 1380.834,A 0.000,B 0.000,C 90.000,E1 6.144} C_DIS
LIN {X -0.159,Y -393.884,Z 1380.832,A 0.000,B 0.000,C 90.000,E1 5.739} C_DIS
LIN {X -0.162,Y -398.460,Z 1380.830,A 0.000,B 0.000,C 90.000,E1 5.334} C_DIS
LIN {X 0.159,Y -406.100,Z 1380.826,A 0.000,B 0.000,C 90.000,E1 4.702} C_DIS
LIN {X -0.189,Y -410.643,Z 1380.824,A 0.000,B 0.000,C 90.000,E1 4.359} C_DIS
LIN {X 0.076,Y -414.971,Z 1380.822,A 0.000,B 0.000,C 90.000,E1 3.898} C_DIS
LIN {X -0.057,Y -417.917,Z 1380.820,A 0.000,B 0.000,C 90.000,E1 3.612} C_DIS
LIN {X -0.160,Y -421.814,Z 1380.817,A 0.000,B 0.000,C 90.000,E1 3.151} C_DIS
LIN {X -0.022,Y -424.617,Z 1380.816,A 0.000,B 0.000,C 90.000,E1 2.808} C_DIS
LIN {X -0.176,Y -432.045,Z 1380.810,A 0.000,B 0.000,C 90.000,E1 1.833} C_DIS
LIN {X 0.091,Y -437.898,Z 1380.806,A 0.000,B 0.000,C 90.000,E1 0.974} C_DIS
LIN {X 0.000,Y -444.515,Z 1380.800,A 0.000,B 0.000,C 90.000,E1 360.000} C_DIS
LIN {X 0.003,Y -449.941,Z 1380.795,A 0.000,B 0.000,C 90.000,E1 359.141} C_DIS
LIN {X -0.134,Y -453.892,Z 1380.792,A 0.000,B 0.000,C 90.000,E1 358.511} C_DIS
LIN {X -0.135,Y -458.427,Z 1380.787,A 0.000,B 0.000,C 90.000,E1 357.707} C_DIS
LIN {X -0.114,Y -462.594,Z 1380.783,A 0.000,B 0.000,C 90.000,E1 356.906} C_DIS
LIN {X -0.028,Y -466.519,Z 1380.778,A 0.000,B 0.000,C 90.000,E1 356.102} C_DIS
LIN {X -0.100,Y -471.380,Z 1380.772,A 0.000,B 0.000,C 90.000,E1 355.008} C_DIS
LIN {X -0.049,Y -473.980,Z 1380.769,A 0.000,B 0.000,C 90.000,E1 354.375} C_DIS
LIN {X -0.148,Y -477.554,Z 1380.764,A 0.000,B 0.000,C 90.000,E1 353.451} C_DIS
LIN {X -0.209,Y -480.846,Z 1380.758,A 0.000,B 0.000,C 90.000,E1 352.527} C_DIS
LIN {X 0.244,Y -483.729,Z 1380.753,A 0.000,B 0.000,C 90.000,E1 351.546} C_DIS
LIN {X -0.102,Y -485.514,Z 1380.750,A 0.000,B 0.000,C 90.000,E1 350.971} C_DIS
LIN {X 0.121,Y -486.976,Z 1380.746,A 0.000,B 0.000,C 90.000,E1 350.330} C_DIS
LIN {X -0.004,Y -487.355,Z 1380.745,A 0.000,B 0.000,C 90.000,E1 350.038} C_DIS
LIN {X -0.124,Y -487.508,Z 1380.743,A 0.000,B 0.000,C 90.000,E1 349.746} C_DIS
LIN {X 0.236,Y -487.289,Z 1380.741,A 0.000,B 0.000,C 90.000,E1 349.398} C_DIS
LIN {X 0.117,Y -486.097,Z 1380.740,A 0.000,B 0.000,C 90.000,E1 349.106} C_DIS
LIN {X 0.169,Y -484.246,Z 1380.739,A 0.000,B 0.000,C 90.000,E1 348.993} C_DIS
LIN {X -0.106,Y -447.059,Z 1380.734,A 0.000,B 0.000,C 90.000,E1 348.117} C_DIS
LIN {X 0.159,Y -411.609,Z 1380.728,A 0.000,B 0.000,C 90.000,E1 347.061} C_DIS
LIN {X 0.103,Y -379.879,Z 1380.722,A 0.000,B 0.000,C 90.000,E1 345.992} C_DIS
LIN {X -0.052,Y -359.595,Z 1380.718,A 0.000,B 0.000,C 90.000,E1 345.227} C_DIS
LIN {X -0.081,Y -359.531,Z 1380.718,A 0.000,B 0.000,C 90.000,E1 345.227} C_DIS
LIN {X -0.107,Y -361.978,Z 1380.682,A 0.000,B 0.000,C 90.000,E1 338.827} C_DIS
LIN {X 0.001,Y -365.933,Z 1380.643,A 0.000,B 0.000,C 90.000,E1 331.719} C_DIS
LIN {X 0.079,Y -366.221,Z 1380.641,A 0.000,B 0.000,C 90.000,E1 331.335} C_DIS
LIN {X -0.024,Y -371.300,Z 1380.604,A 0.000,B 0.000,C 90.000,E1 324.689} C_DIS
LIN {X -0.035,Y -371.728,Z 1380.602,A 0.000,B 0.000,C 90.000,E1 324.322} C_DIS
LIN {X 0.043,Y -377.298,Z 1380.567,A 0.000,B 0.000,C 90.000,E1 318.081} C_DIS
LIN {X -0.211,Y -378.205,Z 1380.563,A 0.000,B 0.000,C 90.000,E1 317.391} C_DIS
LIN {X 0.061,Y -383.877,Z 1380.531,A 0.000,B 0.000,C 90.000,E1 311.553} C_DIS
LIN {X 0.110,Y -384.854,Z 1380.527,A 0.000,B 0.000,C 90.000,E1 310.825} C_DIS
LIN {X 0.032,Y -390.548,Z 1380.495,A 0.000,B 0.000,C 90.000,E1 305.105} C_DIS
LIN {X 0.099,Y -391.039,Z 1380.493,A 0.000,B 0.000,C 90.000,E1 304.739} C_DIS
LIN {X -0.055,Y -391.402,Z 1380.491,A 0.000,B 0.000,C 90.000,E1 304.405} C_DIS
LIN {X -0.111,Y -396.766,Z 1380.460,A 0.000,B 0.000,C 90.000,E1 298.743} C_DIS
LIN {X 0.107,Y -397.100,Z 1380.458,A 0.000,B 0.000,C 90.000,E1 298.359} C_DIS
LIN {X -0.107,Y -401.554,Z 1380.427,A 0.000,B 0.000,C 90.000,E1 292.770} C_DIS
LIN {X 0.034,Y -404.618,Z 1380.395,A 0.000,B 0.000,C 90.000,E1 287.166} C_DIS
LIN {X 0.137,Y -404.756,Z 1380.394,A 0.000,B 0.000,C 90.000,E1 286.804} C_DIS
LIN {X 0.136,Y -406.073,Z 1380.365,A 0.000,B 0.000,C 90.000,E1 281.591} C_DIS
LIN {X 0.144,Y -406.113,Z 1380.363,A 0.000,B 0.000,C 90.000,E1 281.243} C_DIS
LIN {X 0.179,Y -405.669,Z 1380.334,A 0.000,B 0.000,C 90.000,E1 276.030} C_DIS
LIN {X 0.184,Y -405.558,Z 1380.332,A 0.000,B 0.000,C 90.000,E1 275.682} C_DIS
LIN {X -0.145,Y -403.524,Z 1380.305,A 0.000,B 0.000,C 90.000,E1 270.859} C_DIS
LIN {X -0.178,Y -403.315,Z 1380.303,A 0.000,B 0.000,C 90.000,E1 270.516} C_DIS
LIN {X 0.011,Y -398.972,Z 1380.272,A 0.000,B 0.000,C 90.000,E1 264.894} C_DIS
LIN {X -0.183,Y -393.144,Z 1380.242,A 0.000,B 0.000,C 90.000,E1 259.634} C_DIS
LIN {X -0.151,Y -392.878,Z 1380.240,A 0.000,B 0.000,C 90.000,E1 259.275} C_DIS
LIN {X -0.129,Y -386.042,Z 1380.213,A 0.000,B 0.000,C 90.000,E1 254.283} C_DIS
LIN {X -0.082,Y -385.313,Z 1380.209,A 0.000,B 0.000,C 90.000,E1 253.559} C_DIS
LIN {X -0.060,Y -384.854,Z 1380.207,A 0.000,B 0.000,C 90.000,E1 253.196} C_DIS
LIN {X 0.042,Y -378.033,Z 1380.183,A 0.000,B 0.000,C 90.000,E1 248.847} C_DIS
LIN {X -0.081,Y -376.285,Z 1380.174,A 0.000,B 0.000,C 90.000,E1 247.411} C_DIS
LIN {X -0.102,Y -375.731,Z 1380.172,A 0.000,B 0.000,C 90.000,E1 247.050} C_DIS
LIN {X 0.002,Y -368.994,Z 1380.150,A 0.000,B 0.000,C 90.000,E1 242.999} C_DIS
LIN {X -0.095,Y -366.135,Z 1380.138,A 0.000,B 0.000,C 90.000,E1 240.795} C_DIS
LIN {X -0.189,Y -359.265,Z 1380.115,A 0.000,B 0.000,C 90.000,E1 236.707} C_DIS
LIN {X 0.037,Y -355.926,Z 1380.100,A 0.000,B 0.000,C 90.000,E1 234.036} C_DIS
LIN {X 0.128,Y -348.857,Z 1380.075,A 0.000,B 0.000,C 90.000,E1 229.461} C_DIS
LIN {X -0.032,Y -346.235,Z 1380.062,A 0.000,B 0.000,C 90.000,E1 227.187} C_DIS
LIN {X 0.091,Y -345.765,Z 1380.060,A 0.000,B 0.000,C 90.000,E1 226.782} C_DIS
LIN {X 0.051,Y -339.036,Z 1380.032,A 0.000,B 0.000,C 90.000,E1 221.757} C_DIS
LIN {X -0.082,Y -336.890,Z 1380.019,A 0.000,B 0.000,C 90.000,E1 219.439} C_DIS
LIN {X -0.067,Y -331.223,Z 1379.991,A 0.000,B 0.000,C 90.000,E1 214.326} C_DIS
LIN {X -0.009,Y -329.324,Z 1379.975,A 0.000,B 0.000,C 90.000,E1 211.544} C_DIS
LIN {X 0.012,Y -326.426,Z 1379.958,A 0.000,B 0.000,C 90.000,E1 208.359} C_DIS
LIN {X 0.042,Y -323.850,Z 1379.929,A 0.000,B 0.000,C 90.000,E1 203.153} C_DIS
LIN {X -0.024,Y -321.162,Z 1379.895,A 0.000,B 0.000,C 90.000,E1 197.040} C_DIS
LIN {X -0.042,Y -321.177,Z 1379.895,A 0.000,B 0.000,C 90.000,E1 197.040} C_DIS
LIN {X 0.088,Y -345.048,Z 1379.888,A 0.000,B 0.000,C 90.000,E1 195.843} C_DIS
LIN {X -0.053,Y -372.133,Z 1379.882,A 0.000,B 0.000,C 90.000,E1 194.717} C_DIS
LIN {X 0.059,Y -399.391,Z 1379.876,A 0.000,B 0.000,C 90.000,E1 193.703} C_DIS
LIN {X 0.215,Y -432.283,Z 1379.870,A 0.000,B 0.000,C 90.000,E1 192.647} C_DIS
LIN {X -0.101,Y -439.350,Z 1379.869,A 0.000,B 0.000,C 90.000,E1 192.479} C_DIS
LIN {X 0.011,Y -440.524,Z 1379.869,A 0.000,B 0.000,C 90.000,E1 192.355} C_DIS
LIN {X 0.106,Y -441.857,Z 1379.867,A 0.000,B 0.000,C 90.000,E1 192.063} C_DIS
LIN {X -0.174,Y -442.650,Z 1379.865,A 0.000,B 0.000,C 90.000,E1 191.771} C_DIS
LIN {X -0.014,Y -442.992,Z 1379.864,A 0.000,B 0.000,C 90.000,E1 191.422} C_DIS
LIN {X 0.150,Y -443.131,Z 1379.862,A 0.000,B 0.000,C 90.000,E1 191.074} C_DIS
LIN {X -0.055,Y -442.980,Z 1379.854,A 0.000,B 0.000,C 90.000,E1 189.792} C_DIS
LIN {X 0.061,Y -442.722,Z 1379.844,A 0.000,B 0.000,C 90.000,E1 187.814} C_DIS
LIN {X -0.118,Y -442.454,Z 1379.834,A 0.000,B 0.000,C 90.000,E1 186.201} C_DIS
LIN {X -0.014,Y -442.108,Z 1379.827,A 0.000,B 0.000,C 90.000,E1 184.878} C_DIS
LIN {X -0.183,Y -441.824,Z 1379.823,A 0.000,B 0.000,C 90.000,E1 184.245} C_DIS
LIN {X 0.084,Y -441.378,Z 1379.820,A 0.000,B 0.000,C 90.000,E1 183.555} C_DIS
LIN {X 0.021,Y -440.353,Z 1379.814,A 0.000,B 0.000,C 90.000,E1 182.579} C_DIS
LIN {X 0.057,Y -438.747,Z 1379.807,A 0.000,B 0.000,C 90.000,E1 181.260} C_DIS
LIN {X 0.055,Y -436.410,Z 1379.800,A 0.000,B 0.000,C 90.000,E1 179.943} C_DIS
LIN {X 0.158,Y -435.782,Z 1379.798,A 0.000,B 0.000,C 90.000,E1 179.599} C_DIS
LIN {X 0.016,Y -433.292,Z 1379.792,A 0.000,B 0.000,C 90.000,E1 178.625} C_DIS
LIN {X 0.206,Y -431.400,Z 1379.789,A 0.000,B 0.000,C 90.000,E1 177.936} C_DIS
LIN {X -0.063,Y -429.155,Z 1379.785,A 0.000,B 0.000,C 90.000,E1 177.306} C_DIS
LIN {X 0.065,Y -427.262,Z 1379.782,A 0.000,B 0.000,C 90.000,E1 176.788} C_DIS
LIN {X 0.183,Y -424.548,Z 1379.779,A 0.000,B 0.000,C 90.000,E1 176.102} C_DIS
LIN {X -0.051,Y -419.408,Z 1379.773,A 0.000,B 0.000,C 90.000,E1 175.122} C_DIS
LIN {X 0.035,Y -414.433,Z 1379.768,A 0.000,B 0.000,C 90.000,E1 174.261} C_DIS
LIN {X 0.084,Y -406.423,Z 1379.761,A 0.000,B 0.000,C 90.000,E1 173.053} C_DIS
LIN {X -0.055,Y -390.795,Z 1379.748,A 0.000,B 0.000,C 90.000,E1 170.622} C_DIS
LIN {X -0.147,Y -384.646,Z 1379.742,A 0.000,B 0.000,C 90.000,E1 169.567} C_DIS
LIN {X 0.081,Y -380.790,Z 1379.738,A 0.000,B 0.000,C 90.000,E1 168.814} C_DIS
LIN {X -0.100,Y -377.294,Z 1379.734,A 0.000,B 0.000,C 90.000,E1 168.117} C_DIS
LIN {X 0.087,Y -375.099,Z 1379.730,A 0.000,B 0.000,C 90.000,E1 167.409} C_DIS
LIN {X 0.073,Y -374.653,Z 1379.729,A 0.000,B 0.000,C 90.000,E1 167.229} C_DIS
LIN {X -0.034,Y -374.445,Z 1379.728,A 0.000,B 0.000,C 90.000,E1 166.992} C_DIS
LIN {X -0.058,Y -374.452,Z 1379.728,A 0.000,B 0.000,C 90.000,E1 166.992} C_DIS
LIN {X 0.074,Y -376.035,Z 1379.726,A 0.000,B 0.000,C 90.000,E1 166.589} C_DIS
LIN {X -0.062,Y -381.063,Z 1379.722,A 0.000,B 0.000,C 90.000,E1 165.880} C_DIS
LIN {X 0.021,Y -387.022,Z 1379.718,A 0.000,B 0.000,C 90.000,E1 165.172} C_DIS
LIN {X 0.122,Y -397.793,Z 1379.712,A 0.000,B 0.000,C 90.000,E1 164.047} C_DIS
LIN {X -0.051,Y -416.508,Z 1379.702,A 0.000,B 0.000,C 90.000,E1 162.362} C_DIS
LIN {X -0.039,Y -441.917,Z 1379.691,A 0.000,B 0.000,C 90.000,E1 160.315} C_DIS
LIN {X 0.019,Y -454.425,Z 1379.685,A 0.000,B 0.000,C 90.000,E1 159.337} C_DIS
LIN {X 0.069,Y -463.676,Z 1379.681,A 0.000,B 0.000,C 90.000,E1 158.592} C_DIS
LIN {X -0.020,Y -472.643,Z 1379.677,A 0.000,B 0.000,C 90.000,E1 157.847} C_DIS
LIN {X 0.166,Y -478.536,Z 1379.674,A 0.000,B 0.000,C 90.000,E1 157.305} C_DIS
LIN {X -0.015,Y -484.334,Z 1379.671,A 0.000,B 0.000,C 90.000,E1 156.794} C_DIS
LIN {X -0.025,Y -494.320,Z 1379.666,A 0.000,B 0.000,C 90.000,E1 155.845} C_DIS
LIN {X -0.149,Y -502.414,Z 1379.661,A 0.000,B 0.000,C 90.000,E1 155.025} C_DIS
LIN {X -0.188,Y -507.571,Z 1379.658,A 0.000,B 0.000,C 90.000,E1 154.460} C_DIS
LIN {X -0.069,Y -515.137,Z 1379.653,A 0.000,B 0.000,C 90.000,E1 153.563} C_DIS
LIN {X 0.169,Y -519.914,Z 1379.650,A 0.000,B 0.000,C 90.000,E1 152.948} C_DIS
LIN {X -0.089,Y -523.293,Z 1379.647,A 0.000,B 0.000,C 90.000,E1 152.538} C_DIS
LIN {X -0.104,Y -526.507,Z 1379.645,A 0.000,B 0.000,C 90.000,E1 152.103} C_DIS
LIN {X -0.009,Y -530.250,Z 1379.642,A 0.000,B 0.000,C 90.000,E1 151.513} C_DIS
LIN {X -0.031,Y -534.259,Z 1379.638,A 0.000,B 0.000,C 90.000,E1 150.795} C_DIS
LIN {X 0.123,Y -537.010,Z 1379.635,A 0.000,B 0.000,C 90.000,E1 150.205} C_DIS
LIN {X -0.168,Y -539.426,Z 1379.631,A 0.000,B 0.000,C 90.000,E1 149.665} C_DIS
LIN {X 0.030,Y -542.562,Z 1379.627,A 0.000,B 0.000,C 90.000,E1 148.791} C_DIS
LIN {X 0.241,Y -544.440,Z 1379.624,A 0.000,B 0.000,C 90.000,E1 148.201} C_DIS
LIN {X 0.031,Y -546.662,Z 1379.619,A 0.000,B 0.000,C 90.000,E1 147.375} C_DIS
LIN {X -0.152,Y -548.577,Z 1379.614,A 0.000,B 0.000,C 90.000,E1 146.548} C_DIS
LIN {X 0.141,Y -550.207,Z 1379.609,A 0.000,B 0.000,C 90.000,E1 145.674} C_DIS
LIN {X 0.248,Y -551.096,Z 1379.606,A 0.000,B 0.000,C 90.000,E1 145.102} C_DIS
LIN {X 0.171,Y -552.627,Z 1379.600,A 0.000,B 0.000,C 90.000,E1 143.989} C_DIS
LIN {X -0.272,Y -553.926,Z 1379.592,A 0.000,B 0.000,C 90.000,E1 142.637} C_DIS
LIN {X 0.063,Y -555.125,Z 1379.583,A 0.000,B 0.000,C 90.000,E1 140.928} C_DIS
LIN {X -0.001,Y -555.973,Z 1379.575,A 0.000,B 0.000,C 90.000,E1 139.542} C_DIS
LIN {X -0.049,Y -556.882,Z 1379.566,A 0.000,B 0.000,C 90.000,E1 137.877} C_DIS
LIN {X 0.222,Y -557.465,Z 1379.558,A 0.000,B 0.000,C 90.000,E1 136.458} C_DIS
LIN {X 0.107,Y -557.986,Z 1379.551,A 0.000,B 0.000,C 90.000,E1 135.081} C_DIS
LIN {X 0.070,Y -558.611,Z 1379.541,A 0.000,B 0.000,C 90.000,E1 133.419} C_DIS
LIN {X -0.034,Y -558.982,Z 1379.534,A 0.000,B 0.000,C 90.000,E1 132.043} C_DIS
LIN {X 0.319,Y -559.313,Z 1379.526,A 0.000,B 0.000,C 90.000,E1 130.620} C_DIS
LIN {X 0.078,Y -560.041,Z 1379.515,A 0.000,B 0.000,C 90.000,E1 128.705} C_DIS
LIN {X -0.175,Y -560.473,Z 1379.512,A 0.000,B 0.000,C 90.000,E1 128.177} C_DIS
LIN {X 0.044,Y -560.560,Z 1379.511,A 0.000,B 0.000,C 90.000,E1 128.016} C_DIS
LIN {X -0.277,Y -561.198,Z 1379.510,A 0.000,B 0.000,C 90.000,E1 127.729} C_DIS
LIN {X -0.182,Y -561.549,Z 1379.508,A 0.000,B 0.000,C 90.000,E1 127.443} C_DIS
LIN {X -0.194,Y -562.366,Z 1379.507,A 0.000,B 0.000,C 90.000,E1 127.237} C_DIS
LIN {X -0.084,Y -563.266,Z 1379.506,A 0.000,B 0.000,C 90.000,E1 127.156} C_DIS
LIN {X -0.212,Y -565.115,Z 1379.506,A 0.000,B 0.000,C 90.000,E1 127.076} C_DIS
LIN {X 0.214,Y -567.377,Z 1379.505,A 0.000,B 0.000,C 90.000,E1 126.950} C_DIS
LIN {X -0.144,Y -577.506,Z 1379.504,A 0.000,B 0.000,C 90.000,E1 126.710} C_DIS
LIN {X 0.168,Y -580.700,Z 1379.503,A 0.000,B 0.000,C 90.000,E1 126.583} C_DIS
LIN {X -0.087,Y -583.715,Z 1379.503,A 0.000,B 0.000,C 90.000,E1 126.503} C_DIS
LIN {X -0.035,Y -586.375,Z 1379.502,A 0.000,B 0.000,C 90.000,E1 126.377} C_DIS
LIN {X 0.045,Y -589.389,Z 1379.501,A 0.000,B 0.000,C 90.000,E1 126.217} C_DIS
LIN {X -0.060,Y -595.443,Z 1379.499,A 0.000,B 0.000,C 90.000,E1 125.884} C_DIS
LIN {X -0.294,Y -601.139,Z 1379.497,A 0.000,B 0.000,C 90.000,E1 125.518} C_DIS
LIN {X 0.364,Y -606.614,Z 1379.495,A 0.000,B 0.000,C 90.000,E1 125.025} C_DIS
LIN {X -0.219,Y -610.678,Z 1379.493,A 0.000,B 0.000,C 90.000,E1 124.739} C_DIS
LIN {X 0.068,Y -618.323,Z 1379.489,A 0.000,B 0.000,C 90.000,E1 123.992} C_DIS
LIN {X 0.091,Y -624.390,Z 1379.485,A 0.000,B 0.000,C 90.000,E1 123.372} C_DIS
LIN {X -0.099,Y -631.039,Z 1379.481,A 0.000,B 0.000,C 90.000,E1 122.625} C_DIS
LIN {X -0.247,Y -636.127,Z 1379.478,A 0.000,B 0.000,C 90.000,E1 122.005} C_DIS
LIN {X 0.185,Y -640.798,Z 1379.474,A 0.000,B 0.000,C 90.000,E1 121.337} C_DIS
LIN {X -0.253,Y -644.286,Z 1379.471,A 0.000,B 0.000,C 90.000,E1 120.875} C_DIS
LIN {X 0.256,Y -648.035,Z 1379.468,A 0.000,B 0.000,C 90.000,E1 120.207} C_DIS
LIN {X -0.089,Y -651.304,Z 1379.465,A 0.000,B 0.000,C 90.000,E1 119.617} C_DIS
LIN {X -0.146,Y -653.564,Z 1379.462,A 0.000,B 0.000,C 90.000,E1 119.127} C_DIS
LIN {X -0.045,Y -654.542,Z 1379.460,A 0.000,B 0.000,C 90.000,E1 118.871} C_DIS
LIN {X 0.171,Y -656.206,Z 1379.458,A 0.000,B 0.000,C 90.000,E1 118.359} C_DIS
LIN {X 0.285,Y -656.932,Z 1379.456,A 0.000,B 0.000,C 90.000,E1 118.103} C_DIS
LIN {X -0.058,Y -657.848,Z 1379.454,A 0.000,B 0.000,C 90.000,E1 117.641} C_DIS
LIN {X 0.185,Y -658.536,Z 1379.451,A 0.000,B 0.000,C 90.000,E1 117.129} C_DIS
LIN {X -0.028,Y -658.515,Z 1379.447,A 0.000,B 0.000,C 90.000,E1 116.411} C_DIS
LIN {X -0.067,Y -658.343,Z 1379.444,A 0.000,B 0.000,C 90.000,E1 115.924} C_DIS
LIN {X 0.185,Y -657.874,Z 1379.441,A 0.000,B 0.000,C 90.000,E1 115.412} C_DIS
LIN {X -0.286,Y -657.586,Z 1379.440,A 0.000,B 0.000,C 90.000,E1 115.207} C_DIS
LIN {X -0.044,Y -656.672,Z 1379.437,A 0.000,B 0.000,C 90.000,E1 114.695} C_DIS
LIN {X -0.198,Y -655.839,Z 1379.436,A 0.000,B 0.000,C 90.000,E1 114.463} C_DIS
LIN {X 0.033,Y -653.434,Z 1379.433,A 0.000,B 0.000,C 90.000,E1 113.951} C_DIS
LIN {X 0.087,Y -652.445,Z 1379.432,A 0.000,B 0.000,C 90.000,E1 113.823} C_DIS
LIN {X -0.017,Y -648.943,Z 1379.430,A 0.000,B 0.000,C 90.000,E1 113.462} C_DIS
LIN {X 0.028,Y -647.621,Z 1379.430,A 0.000,B 0.000,C 90.000,E1 113.334} C_DIS
LIN {X 0.075,Y -645.527,Z 1379.429,A 0.000,B 0.000,C 90.000,E1 113.206} C_DIS
LIN {X -0.253,Y -638.628,Z 1379.427,A 0.000,B 0.000,C 90.000,E1 112.898} C_DIS
LIN {X 0.259,Y -632.173,Z 1379.426,A 0.000,B 0.000,C 90.000,E1 112.642} C_DIS
LIN {X -0.235,Y -619.065,Z 1379.424,A 0.000,B 0.000,C 90.000,E1 112.333} C_DIS
LIN {X -0.297,Y -619.071,Z 1379.424,A 0.000,B 0.000,C 90.000,E1 112.333} C_DIS
LIN {X -0.213,Y -626.640,Z 1379.420,A 0.000,B 0.000,C 90.000,E1 111.535} C_DIS
LIN {X 0.060,Y -632.195,Z 1379.416,A 0.000,B 0.000,C 90.000,E1 110.918} C_DIS
LIN {X -0.122,Y -636.490,Z 1379.413,A 0.000,B 0.000,C 90.000,E1 110.429} C_DIS
LIN {X -0.260,Y -641.182,Z 1379.410,A 0.000,B 0.000,C 90.000,E1 109.812} C_DIS
LIN {X 0.058,Y -645.926,Z 1379.406,A 0.000,B 0.000,C 90.000,E1 109.033} C_DIS
LIN {X -0.150,Y -650.780,Z 1379.401,A 0.000,B 0.000,C 90.000,E1 108.181} C_DIS
LIN {X -0.384,Y -653.912,Z 1379.398,A 0.000,B 0.000,C 90.000,E1 107.583} C_DIS
LIN {X 0.190,Y -656.256,Z 1379.395,A 0.000,B 0.000,C 90.000,E1 107.040} C_DIS
LIN {X 0.146,Y -658.242,Z 1379.392,A 0.000,B 0.000,C 90.000,E1 106.551} C_DIS
LIN {X -0.073,Y -659.850,Z 1379.389,A 0.000,B 0.000,C 90.000,E1 106.079} C_DIS
LIN {X -0.177,Y -660.626,Z 1379.388,A 0.000,B 0.000,C 90.000,E1 105.843} C_DIS
LIN {X 0.339,Y -662.314,Z 1379.384,A 0.000,B 0.000,C 90.000,E1 105.064} C_DIS
LIN {X 0.151,Y -663.218,Z 1379.381,A 0.000,B 0.000,C 90.000,E1 104.592} C_DIS
LIN {X -0.120,Y -664.202,Z 1379.377,A 0.000,B 0.000,C 90.000,E1 103.883} C_DIS
LIN {X -0.296,Y -664.682,Z 1379.374,A 0.000,B 0.000,C 90.000,E1 103.411} C_DIS
LIN {X 0.094,Y -664.920,Z 1379.370,A 0.000,B 0.000,C 90.000,E1 102.647} C_DIS
LIN {X -0.079,Y -664.875,Z 1379.368,A 0.000,B 0.000,C 90.000,E1 102.175} C_DIS
LIN {X 0.262,Y -664.657,Z 1379.365,A 0.000,B 0.000,C 90.000,E1 101.658} C_DIS
LIN {X -0.002,Y -663.809,Z 1379.361,A 0.000,B 0.000,C 90.000,E1 100.950} C_DIS
LIN {X -0.308,Y -663.057,Z 1379.358,A 0.000,B 0.000,C 90.000,E1 100.489} C_DIS
LIN {X 0.154,Y -662.078,Z 1379.355,A 0.000,B 0.000,C 90.000,E1 99.962} C_DIS
LIN {X -0.156,Y -660.913,Z 1379.353,A 0.000,B 0.000,C 90.000,E1 99.500} C_DIS
LIN {X 0.073,Y -658.650,Z 1379.349,A 0.000,B 0.000,C 90.000,E1 98.746} C_DIS
LIN {X 0.280,Y -656.014,Z 1379.345,A 0.000,B 0.000,C 90.000,E1 97.992} C_DIS
LIN {X -0.060,Y -653.989,Z 1379.342,A 0.000,B 0.000,C 90.000,E1 97.530} C_DIS
LIN {X -0.191,Y -652.919,Z 1379.340,A 0.000,B 0.000,C 90.000,E1 97.296} C_DIS
LIN {X -0.126,Y -649.234,Z 1379.336,A 0.000,B 0.000,C 90.000,E1 96.549} C_DIS
LIN {X 0.136,Y -646.502,Z 1379.334,A 0.000,B 0.000,C 90.000,E1 96.030} C_DIS
LIN {X 0.078,Y -641.350,Z 1379.329,A 0.000,B 0.000,C 90.000,E1 95.163} C_DIS
LIN {X 0.153,Y -637.409,Z 1379.325,A 0.000,B 0.000,C 90.000,E1 94.531} C_DIS
LIN {X 0.324,Y -633.970,Z 1379.323,A 0.000,B 0.000,C 90.000,E1 94.012} C_DIS
LIN {X -0.203,Y -630.026,Z 1379.320,A 0.000,B 0.000,C 90.000,E1 93.555} C_DIS
LIN {X -0.226,Y -624.326,Z 1379.316,A 0.000,B 0.000,C 90.000,E1 92.922} C_DIS
LIN {X 0.031,Y -616.840,Z 1379.312,A 0.000,B 0.000,C 90.000,E1 92.178} C_DIS
LIN {X 0.257,Y -608.872,Z 1379.308,A 0.000,B 0.000,C 90.000,E1 91.432} C_DIS
LIN {X 0.160,Y -603.251,Z 1379.306,A 0.000,B 0.000,C 90.000,E1 90.974} C_DIS
LIN {X -0.097,Y -597.003,Z 1379.303,A 0.000,B 0.000,C 90.000,E1 90.573} C_DIS
LIN {X 0.254,Y -593.685,Z 1379.302,A 0.000,B 0.000,C 90.000,E1 90.344} C_DIS
LIN {X -0.103,Y -588.509,Z 1379.301,A 0.000,B 0.000,C 90.000,E1 90.115} C_DIS
LIN {X -0.177,Y -583.221,Z 1379.299,A 0.000,B 0.000,C 90.000,E1 89.885} C_DIS
LIN {X -0.156,Y -577.502,Z 1379.298,A 0.000,B 0.000,C 90.000,E1 89.599} C_DIS
LIN {X 0.179,Y -576.406,Z 1379.297,A 0.000,B 0.000,C 90.000,E1 89.484} C_DIS
LIN {X -0.054,Y -574.456,Z 1379.296,A 0.000,B 0.000,C 90.000,E1 89.312} C_DIS
LIN {X -0.131,Y -573.909,Z 1379.296,A 0.000,B 0.000,C 90.000,E1 89.198} C_DIS
LIN {X 0.177,Y -573.669,Z 1379.294,A 0.000,B 0.000,C 90.000,E1 88.854} C_DIS
LIN {X 0.181,Y -574.101,Z 1379.289,A 0.000,B 0.000,C 90.000,E1 88.051} C_DIS
LIN {X 0.256,Y -575.983,Z 1379.277,A 0.000,B 0.000,C 90.000,E1 85.869} C_DIS
LIN {X 0.050,Y -578.470,Z 1379.264,A 0.000,B 0.000,C 90.000,E1 83.451} C_DIS
LIN {X -0.031,Y -580.418,Z 1379.255,A 0.000,B 0.000,C 90.000,E1 81.837} C_DIS
LIN {X 0.092,Y -582.332,Z 1379.246,A 0.000,B 0.000,C 90.000,E1 80.208} C_DIS
LIN {X -0.217,Y -583.575,Z 1379.240,A 0.000,B 0.000,C 90.000,E1 79.162} C_DIS
LIN {X -0.154,Y -584.933,Z 1379.232,A 0.000,B 0.000,C 90.000,E1 77.813} C_DIS
LIN {X 0.177,Y -586.342,Z 1379.223,A 0.000,B 0.000,C 90.000,E1 76.172} C_DIS
LIN {X 0.100,Y -587.529,Z 1379.214,A 0.000,B 0.000,C 90.000,E1 74.574} C_DIS
LIN {X -0.208,Y -588.337,Z 1379.207,A 0.000,B 0.000,C 90.000,E1 73.268} C_DIS
LIN {X 0.085,Y -589.259,Z 1379.198,A 0.000,B 0.000,C 90.000,E1 71.638} C_DIS
LIN {X -0.155,Y -590.208,Z 1379.189,A 0.000,B 0.000,C 90.000,E1 70.061} C_DIS
LIN {X -0.177,Y -591.589,Z 1379.176,A 0.000,B 0.000,C 90.000,E1 67.667} C_DIS
LIN {X -0.047,Y -592.942,Z 1379.166,A 0.000,B 0.000,C 90.000,E1 65.793} C_DIS
LIN {X -0.079,Y -594.302,Z 1379.157,A 0.000,B 0.000,C 90.000,E1 64.204} C_DIS
LIN {X -0.087,Y -595.493,Z 1379.148,A 0.000,B 0.000,C 90.000,E1 62.615} C_DIS
LIN {X 0.135,Y -597.830,Z 1379.133,A 0.000,B 0.000,C 90.000,E1 59.950} C_DIS
LIN {X -0.059,Y -599.552,Z 1379.123,A 0.000,B 0.000,C 90.000,E1 58.122} C_DIS
LIN {X -0.205,Y -601.298,Z 1379.113,A 0.000,B 0.000,C 90.000,E1 56.294} C_DIS
LIN {X -0.230,Y -603.157,Z 1379.101,A 0.000,B 0.000,C 90.000,E1 54.196} C_DIS
LIN {X -0.116,Y -604.819,Z 1379.091,A 0.000,B 0.000,C 90.000,E1 52.351} C_DIS
LIN {X -0.017,Y -605.604,Z 1379.085,A 0.000,B 0.000,C 90.000,E1 51.295} C_DIS
LIN {X -0.018,Y -606.282,Z 1379.078,A 0.000,B 0.000,C 90.000,E1 49.989} C_DIS
LIN {X 0.174,Y -606.955,Z 1379.069,A 0.000,B 0.000,C 90.000,E1 48.405} C_DIS
LIN {X 0.110,Y -607.275,Z 1379.062,A 0.000,B 0.000,C 90.000,E1 47.106} C_DIS
LIN {X 0.023,Y -607.360,Z 1379.055,A 0.000,B 0.000,C 90.000,E1 45.810} C_DIS
LIN {X 0.321,Y -607.378,Z 1379.050,A 0.000,B 0.000,C 90.000,E1 45.000} C_DIS
LIN {X 0.241,Y -607.030,Z 1379.043,A 0.000,B 0.000,C 90.000,E1 43.704} C_DIS
LIN {X -0.269,Y -606.462,Z 1379.036,A 0.000,B 0.000,C 90.000,E1 42.447} C_DIS
LIN {X -0.338,Y -605.789,Z 1379.028,A 0.000,B 0.000,C 90.000,E1 41.148} C_DIS
LIN {X 0.041,Y -604.931,Z 1379.021,A 0.000,B 0.000,C 90.000,E1 39.806} C_DIS
LIN {X 0.146,Y -604.094,Z 1379.015,A 0.000,B 0.000,C 90.000,E1 38.749} C_DIS
LIN {X -0.143,Y -603.117,Z 1379.010,A 0.000,B 0.000,C 90.000,E1 37.729} C_DIS
LIN {X 0.035,Y -601.896,Z 1379.004,A 0.000,B 0.000,C 90.000,E1 36.664} C_DIS
LIN {X -0.051,Y -600.823,Z 1378.999,A 0.000,B 0.000,C 90.000,E1 35.884} C_DIS
LIN {X -0.148,Y -599.502,Z 1378.995,A 0.000,B 0.000,C 90.000,E1 35.105} C_DIS
LIN {X -0.006,Y -598.451,Z 1378.992,A 0.000,B 0.000,C 90.000,E1 34.565} C_DIS
LIN {X -0.002,Y -595.529,Z 1378.985,A 0.000,B 0.000,C 90.000,E1 33.245} C_DIS
LIN {X 0.120,Y -594.210,Z 1378.982,A 0.000,B 0.000,C 90.000,E1 32.704} C_DIS
LIN {X -0.169,Y -591.310,Z 1378.976,A 0.000,B 0.000,C 90.000,E1 31.671} C_DIS
LIN {X -0.079,Y -589.730,Z 1378.973,A 0.000,B 0.000,C 90.000,E1 31.131} C_DIS
LIN {X -0.117,Y -586.862,Z 1378.969,A 0.000,B 0.000,C 90.000,E1 30.335} C_DIS
LIN {X -0.184,Y -583.652,Z 1378.964,A 0.000,B 0.000,C 90.000,E1 29.539} C_DIS
LIN {X -0.154,Y -581.322,Z 1378.961,A 0.000,B 0.000,C 90.000,E1 28.999} C_DIS
LIN {X 0.221,Y -577.581,Z 1378.957,A 0.000,B 0.000,C 90.000,E1 28.153} C_DIS
LIN {X 0.127,Y -571.919,Z 1378.951,A 0.000,B 0.000,C 90.000,E1 27.078} C_DIS
LIN {X 0.303,Y -566.379,Z 1378.945,A 0.000,B 0.000,C 90.000,E1 26.104} C_DIS
LIN {X -0.252,Y -561.263,Z 1378.941,A 0.000,B 0.000,C 90.000,E1 25.335} C_DIS
LIN {X -0.141,Y -557.593,Z 1378.938,A 0.000,B 0.000,C 90.000,E1 24.771} C_DIS
LIN {X -0.155,Y -552.674,Z 1378.934,A 0.000,B 0.000,C 90.000,E1 24.079} C_DIS
LIN {X 0.010,Y -549.592,Z 1378.931,A 0.000,B 0.000,C 90.000,E1 23.643} C_DIS
LIN {X 0.035,Y -545.159,Z 1378.928,A 0.000,B 0.000,C 90.000,E1 23.078} C_DIS
LIN {X -0.140,Y -538.220,Z 1378.924,A 0.000,B 0.000,C 90.000,E1 22.259} C_DIS
LIN {X -0.045,Y -531.994,Z 1378.920,A 0.000,B 0.000,C 90.000,E1 21.535} C_DIS
LIN {X -0.160,Y -521.650,Z 1378.913,A 0.000,B 0.000,C 90.000,E1 20.429} C_DIS
LIN {X -0.093,Y -512.454,Z 1378.908,A 0.000,B 0.000,C 90.000,E1 19.450} C_DIS
LIN {X -0.081,Y -503.090,Z 1378.903,A 0.000,B 0.000,C 90.000,E1 18.489} C_DIS
LIN {X -0.205,Y -492.165,Z 1378.897,A 0.000,B 0.000,C 90.000,E1 17.402} C_DIS
LIN {X 0.005,Y -479.865,Z 1378.890,A 0.000,B 0.000,C 90.000,E1 16.134} C_DIS
LIN {X -0.001,Y -465.986,Z 1378.882,A 0.000,B 0.000,C 90.000,E1 14.717} C_DIS
LIN {X 0.029,Y -454.987,Z 1378.876,A 0.000,B 0.000,C 90.000,E1 13.592} C_DIS
LIN {X 0.027,Y -438.241,Z 1378.866,A 0.000,B 0.000,C 90.000,E1 11.827} C_DIS
LIN {X -0.006,Y -420.220,Z 1378.854,A 0.000,B 0.000,C 90.000,E1 9.792} C_DIS
LIN {X -0.148,Y -409.277,Z 1378.847,A 0.000,B 0.000,C 90.000,E1 8.511} C_DIS
LIN {X 0.139,Y -400.763,Z 1378.842,A 0.000,B 0.000,C 90.000,E1 7.473} C_DIS
LIN {X -0.053,Y -396.657,Z 1378.839,A 0.000,B 0.000,C 90.000,E1 7.004} C_DIS
LIN {X -0.064,Y -392.808,Z 1378.836,A 0.000,B 0.000,C 90.000,E1 6.486} C_DIS
LIN {X 0.107,Y -391.408,Z 1378.835,A 0.000,B 0.000,C 90.000,E1 6.201} C_DIS
LIN {X -0.188,Y -391.210,Z 1378.834,A 0.000,B 0.000,C 90.000,E1 6.201} C_DIS
LIN {X 0.164,Y -391.230,Z 1378.834,A 0.000,B 0.000,C 90.000,E1 6.144} C_DIS
LIN {X -0.148,Y -394.173,Z 1378.832,A 0.000,B 0.000,C 90.000,E1 5.796} C_DIS
LIN {X -0.111,Y -399.422,Z 1378.830,A 0.000,B 0.000,C 90.000,E1 5.334} C_DIS
LIN {X -0.082,Y -406.885,Z 1378.826,A 0.000,B 0.000,C 90.000,E1 4.759} C_DIS
LIN {X 0.066,Y -411.375,Z 1378.824,A 0.000,B 0.000,C 90.000,E1 4.359} C_DIS
LIN {X 0.127,Y -417.150,Z 1378.821,A 0.000,B 0.000,C 90.000,E1 3.784} C_DIS
LIN {X -0.178,Y -424.074,Z 1378.817,A 0.000,B 0.000,C 90.000,E1 3.037} C_DIS
LIN {X -0.081,Y -431.436,Z 1378.811,A 0.000,B 0.000,C 90.000,E1 2.064} C_DIS
LIN {X -0.142,Y -439.726,Z 1378.805,A 0.000,B 0.000,C 90.000,E1 0.917} C_DIS
LIN {X 0.000,Y -445.832,Z 1378.800,A 0.000,B 0.000,C 90.000,E1 360.000} C_DIS
LIN {X 0.013,Y -451.276,Z 1378.795,A 0.000,B 0.000,C 90.000,E1 359.141} C_DIS
LIN {X -0.026,Y -456.156,Z 1378.791,A 0.000,B 0.000,C 90.000,E1 358.339} C_DIS
LIN {X -0.101,Y -459.812,Z 1378.787,A 0.000,B 0.000,C 90.000,E1 357.707} C_DIS
LIN {X 0.066,Y -464.781,Z 1378.782,A 0.000,B 0.000,C 90.000,E1 356.731} C_DIS
LIN {X 0.035,Y -467.903,Z 1378.778,A 0.000,B 0.000,C 90.000,E1 356.102} C_DIS
LIN {X -0.019,Y -472.798,Z 1378.772,A 0.000,B 0.000,C 90.000,E1 355.008} C_DIS
LIN {X 0.045,Y -475.377,Z 1378.769,A 0.000,B 0.000,C 90.000,E1 354.375} C_DIS
LIN {X 0.127,Y -477.795,Z 1378.765,A 0.000,B 0.000,C 90.000,E1 353.742} C_DIS
LIN {X 0.067,Y -481.156,Z 1378.760,A 0.000,B 0.000,C 90.000,E1 352.818} C_DIS
LIN {X 0.186,Y -483.204,Z 1378.757,A 0.000,B 0.000,C 90.000,E1 352.186} C_DIS
LIN {X 0.256,Y -486.003,Z 1378.752,A 0.000,B 0.000,C 90.000,E1 351.254} C_DIS
LIN {X -0.196,Y -488.547,Z 1378.746,A 0.000,B 0.000,C 90.000,E1 350.387} C_DIS
LIN {X 0.053,Y -489.872,Z 1378.743,A 0.000,B 0.000,C 90.000,E1 349.746} C_DIS
LIN {X -0.060,Y -490.316,Z 1378.741,A 0.000,B 0.000,C 90.000,E1 349.454} C_DIS
LIN {X -0.169,Y -490.541,Z 1378.740,A 0.000,B 0.000,C 90.000,E1 349.162} C_DIS
LIN {X 0.204,Y -490.459,Z 1378.738,A 0.000,B 0.000,C 90.000,E1 348.814} C_DIS
LIN {X 0.096,Y -489.732,Z 1378.736,A 0.000,B 0.000,C 90.000,E1 348.522} C_DIS
LIN {X -0.246,Y -488.718,Z 1378.735,A 0.000,B 0.000,C 90.000,E1 348.409} C_DIS
LIN {X 0.160,Y -487.027,Z 1378.735,A 0.000,B 0.000,C 90.000,E1 348.285} C_DIS
LIN {X 0.006,Y -448.346,Z 1378.729,A 0.000,B 0.000,C 90.000,E1 347.297} C_DIS
LIN {X -0.169,Y -416.536,Z 1378.724,A 0.000,B 0.000,C 90.000,E1 346.353} C_DIS
LIN {X 0.011,Y -388.407,Z 1378.719,A 0.000,B 0.000,C 90.000,E1 345.338} C_DIS
LIN {X -0.072,Y -360.448,Z 1378.712,A 0.000,B 0.000,C 90.000,E1 344.212} C_DIS
LIN {X 0.063,Y -359.681,Z 1378.712,A 0.000,B 0.000,C 90.000,E1 344.157} C_DIS
LIN {X 0.032,Y -359.624,Z 1378.712,A 0.000,B 0.000,C 90.000,E1 344.157} C_DIS
LIN {X 0.138,Y -361.981,Z 1378.682,A 0.000,B 0.000,C 90.000,E1 338.773} C_DIS
LIN {X -0.092,Y -365.947,Z 1378.643,A 0.000,B 0.000,C 90.000,E1 331.719} C_DIS
LIN {X 0.162,Y -366.226,Z 1378.641,A 0.000,B 0.000,C 90.000,E1 331.307} C_DIS
LIN {X -0.117,Y -371.317,Z 1378.604,A 0.000,B 0.000,C 90.000,E1 324.689} C_DIS
LIN {X 0.174,Y -371.740,Z 1378.602,A 0.000,B 0.000,C 90.000,E1 324.276} C_DIS
LIN {X -0.038,Y -377.789,Z 1378.565,A 0.000,B 0.000,C 90.000,E1 317.715} C_DIS
LIN {X 0.230,Y -378.214,Z 1378.563,A 0.000,B 0.000,C 90.000,E1 317.310} C_DIS
LIN {X -0.033,Y -383.896,Z 1378.531,A 0.000,B 0.000,C 90.000,E1 311.553} C_DIS
LIN {X 0.015,Y -384.867,Z 1378.527,A 0.000,B 0.000,C 90.000,E1 310.825} C_DIS
LIN {X -0.062,Y -390.566,Z 1378.495,A 0.000,B 0.000,C 90.000,E1 305.105} C_DIS
LIN {X 0.004,Y -391.059,Z 1378.493,A 0.000,B 0.000,C 90.000,E1 304.739} C_DIS
LIN {X -0.150,Y -391.410,Z 1378.491,A 0.000,B 0.000,C 90.000,E1 304.405} C_DIS
LIN {X 0.142,Y -396.783,Z 1378.460,A 0.000,B 0.000,C 90.000,E1 298.693} C_DIS
LIN {X 0.012,Y -397.106,Z 1378.458,A 0.000,B 0.000,C 90.000,E1 298.359} C_DIS
LIN {X -0.203,Y -401.568,Z 1378.426,A 0.000,B 0.000,C 90.000,E1 292.770} C_DIS
LIN {X -0.061,Y -404.631,Z 1378.395,A 0.000,B 0.000,C 90.000,E1 287.166} C_DIS
LIN {X 0.041,Y -404.754,Z 1378.393,A 0.000,B 0.000,C 90.000,E1 286.804} C_DIS
LIN {X 0.039,Y -406.081,Z 1378.365,A 0.000,B 0.000,C 90.000,E1 281.591} C_DIS
LIN {X 0.047,Y -406.107,Z 1378.363,A 0.000,B 0.000,C 90.000,E1 281.243} C_DIS
LIN {X 0.083,Y -405.672,Z 1378.334,A 0.000,B 0.000,C 90.000,E1 276.030} C_DIS
LIN {X 0.092,Y -405.305,Z 1378.330,A 0.000,B 0.000,C 90.000,E1 275.334} C_DIS
LIN {X 0.162,Y -403.516,Z 1378.305,A 0.000,B 0.000,C 90.000,E1 270.802} C_DIS
LIN {X 0.130,Y -403.307,Z 1378.303,A 0.000,B 0.000,C 90.000,E1 270.458} C_DIS
LIN {X -0.085,Y -398.961,Z 1378.272,A 0.000,B 0.000,C 90.000,E1 264.894} C_DIS
LIN {X 0.109,Y -393.133,Z 1378.242,A 0.000,B 0.000,C 90.000,E1 259.577} C_DIS
LIN {X 0.141,Y -392.867,Z 1378.240,A 0.000,B 0.000,C 90.000,E1 259.218} C_DIS
LIN {X -0.118,Y -386.028,Z 1378.213,A 0.000,B 0.000,C 90.000,E1 254.267} C_DIS
LIN {X -0.176,Y -385.299,Z 1378.209,A 0.000,B 0.000,C 90.000,E1 253.559} C_DIS
LIN {X -0.154,Y -384.828,Z 1378.207,A 0.000,B 0.000,C 90.000,E1 253.196} C_DIS
LIN {X -0.050,Y -378.015,Z 1378.182,A 0.000,B 0.000,C 90.000,E1 248.847} C_DIS
LIN {X 0.173,Y -376.270,Z 1378.174,A 0.000,B 0.000,C 90.000,E1 247.358} C_DIS
LIN {X -0.195,Y -375.704,Z 1378.172,A 0.000,B 0.000,C 90.000,E1 247.050} C_DIS
LIN {X -0.091,Y -368.974,Z 1378.150,A 0.000,B 0.000,C 90.000,E1 242.999} C_DIS
LIN {X -0.187,Y -366.110,Z 1378.138,A 0.000,B 0.000,C 90.000,E1 240.795} C_DIS
LIN {X 0.217,Y -359.244,Z 1378.115,A 0.000,B 0.000,C 90.000,E1 236.628} C_DIS
LIN {X -0.054,Y -355.902,Z 1378.100,A 0.000,B 0.000,C 90.000,E1 234.036} C_DIS
LIN {X 0.038,Y -348.837,Z 1378.075,A 0.000,B 0.000,C 90.000,E1 229.461} C_DIS
LIN {X 0.114,Y -346.220,Z 1378.062,A 0.000,B 0.000,C 90.000,E1 227.148} C_DIS
LIN {X 0.000,Y -345.740,Z 1378.060,A 0.000,B 0.000,C 90.000,E1 226.782} C_DIS
LIN {X -0.039,Y -339.020,Z 1378.032,A 0.000,B 0.000,C 90.000,E1 221.757} C_DIS
LIN {X 0.042,Y -336.876,Z 1378.019,A 0.000,B 0.000,C 90.000,E1 219.402} C_DIS
LIN {X -0.156,Y -331.210,Z 1377.991,A 0.000,B 0.000,C 90.000,E1 214.326} C_DIS
LIN {X -0.097,Y -329.315,Z 1377.975,A 0.000,B 0.000,C 90.000,E1 211.544} C_DIS
LIN {X -0.151,Y -324.884,Z 1377.944,A 0.000,B 0.000,C 90.000,E1 205.976} C_DIS
LIN {X 0.081,Y -323.846,Z 1377.929,A 0.000,B 0.000,C 90.000,E1 203.131} C_DIS
LIN {X 0.140,Y -321.390,Z 1377.901,A 0.000,B 0.000,C 90.000,E1 198.181} C_DIS
LIN {X 0.122,Y -321.429,Z 1377.901,A 0.000,B 0.000,C 90.000,E1 198.181} C_DIS
LIN {X 0.027,Y -344.379,Z 1377.894,A 0.000,B 0.000,C 90.000,E1 196.985} C_DIS
LIN {X -0.054,Y -369.525,Z 1377.888,A 0.000,B 0.000,C 90.000,E1 195.843} C_DIS
LIN {X -0.189,Y -398.414,Z 1377.882,A 0.000,B 0.000,C 90.000,E1 194.717} C_DIS
LIN {X -0.087,Y -431.142,Z 1377.875,A 0.000,B 0.000,C 90.000,E1 193.592} C_DIS
LIN {X -0.001,Y -438.439,Z 1377.874,A 0.000,B 0.000,C 90.000,E1 193.355} C_DIS
LIN {X 0.014,Y -441.207,Z 1377.874,A 0.000,B 0.000,C 90.000,E1 193.244} C_DIS
LIN {X -0.103,Y -442.320,Z 1377.873,A 0.000,B 0.000,C 90.000,E1 193.119} C_DIS
LIN {X 0.023,Y -443.068,Z 1377.872,A 0.000,B 0.000,C 90.000,E1 192.939} C_DIS
LIN {X 0.051,Y -443.581,Z 1377.871,A 0.000,B 0.000,C 90.000,E1 192.771} C_DIS
LIN {X -0.220,Y -444.253,Z 1377.869,A 0.000,B 0.000,C 90.000,E1 192.479} C_DIS
LIN {X 0.040,Y -444.633,Z 1377.867,A 0.000,B 0.000,C 90.000,E1 192.119} C_DIS
LIN {X 0.208,Y -444.813,Z 1377.866,A 0.000,B 0.000,C 90.000,E1 191.771} C_DIS
LIN {X -0.148,Y -444.896,Z 1377.860,A 0.000,B 0.000,C 90.000,E1 190.838} C_DIS
LIN {X -0.155,Y -444.786,Z 1377.851,A 0.000,B 0.000,C 90.000,E1 189.208} C_DIS
LIN {X -0.063,Y -444.632,Z 1377.840,A 0.000,B 0.000,C 90.000,E1 187.239} C_DIS
LIN {X -0.202,Y -444.394,Z 1377.831,A 0.000,B 0.000,C 90.000,E1 185.625} C_DIS
LIN {X -0.192,Y -444.197,Z 1377.826,A 0.000,B 0.000,C 90.000,E1 184.645} C_DIS
LIN {X 0.219,Y -443.700,Z 1377.820,A 0.000,B 0.000,C 90.000,E1 183.612} C_DIS
LIN {X 0.184,Y -442.866,Z 1377.815,A 0.000,B 0.000,C 90.000,E1 182.636} C_DIS
LIN {X 0.135,Y -441.718,Z 1377.809,A 0.000,B 0.000,C 90.000,E1 181.661} C_DIS
LIN {X -0.061,Y -440.807,Z 1377.806,A 0.000,B 0.000,C 90.000,E1 181.031} C_DIS
LIN {X -0.143,Y -439.195,Z 1377.800,A 0.000,B 0.000,C 90.000,E1 180.057} C_DIS
LIN {X 0.085,Y -437.987,Z 1377.797,A 0.000,B 0.000,C 90.000,E1 179.370} C_DIS
LIN {X -0.136,Y -436.510,Z 1377.793,A 0.000,B 0.000,C 90.000,E1 178.740} C_DIS
LIN {X 0.177,Y -433.585,Z 1377.787,A 0.000,B 0.000,C 90.000,E1 177.707} C_DIS
LIN {X -0.038,Y -430.839,Z 1377.783,A 0.000,B 0.000,C 90.000,E1 176.906} C_DIS
LIN {X 0.165,Y -427.367,Z 1377.778,A 0.000,B 0.000,C 90.000,E1 176.045} C_DIS
LIN {X -0.116,Y -424.253,Z 1377.775,A 0.000,B 0.000,C 90.000,E1 175.412} C_DIS
LIN {X 0.056,Y -419.639,Z 1377.770,A 0.000,B 0.000,C 90.000,E1 174.546} C_DIS
LIN {X 0.089,Y -416.517,Z 1377.767,A 0.000,B 0.000,C 90.000,E1 174.033} C_DIS
LIN {X 0.187,Y -412.077,Z 1377.763,A 0.000,B 0.000,C 90.000,E1 173.337} C_DIS
LIN {X 0.184,Y -397.157,Z 1377.751,A 0.000,B 0.000,C 90.000,E1 171.084} C_DIS
LIN {X -0.007,Y -386.630,Z 1377.741,A 0.000,B 0.000,C 90.000,E1 169.342} C_DIS
LIN {X -0.142,Y -381.670,Z 1377.736,A 0.000,B 0.000,C 90.000,E1 168.465} C_DIS
LIN {X -0.136,Y -378.519,Z 1377.732,A 0.000,B 0.000,C 90.000,E1 167.757} C_DIS
LIN {X -0.225,Y -377.804,Z 1377.731,A 0.000,B 0.000,C 90.000,E1 167.589} C_DIS
LIN {X 0.136,Y -377.254,Z 1377.730,A 0.000,B 0.000,C 90.000,E1 167.353} C_DIS
LIN {X 0.082,Y -376.378,Z 1377.726,A 0.000,B 0.000,C 90.000,E1 166.700} C_DIS
LIN {X 0.046,Y -376.384,Z 1377.726,A 0.000,B 0.000,C 90.000,E1 166.700} C_DIS
LIN {X 0.134,Y -376.808,Z 1377.725,A 0.000,B 0.000,C 90.000,E1 166.533} C_DIS
LIN {X 0.097,Y -376.823,Z 1377.725,A 0.000,B 0.000,C 90.000,E1 166.533} C_DIS
LIN {X 0.015,Y -381.214,Z 1377.722,A 0.000,B 0.000,C 90.000,E1 165.880} C_DIS
LIN {X 0.059,Y -386.578,Z 1377.718,A 0.000,B 0.000,C 90.000,E1 165.227} C_DIS
LIN {X 0.167,Y -394.198,Z 1377.714,A 0.000,B 0.000,C 90.000,E1 164.393} C_DIS
LIN {X 0.065,Y -403.474,Z 1377.708,A 0.000,B 0.000,C 90.000,E1 163.504} C_DIS
LIN {X 0.052,Y -418.941,Z 1377.701,A 0.000,B 0.000,C 90.000,E1 162.127} C_DIS
LIN {X 0.068,Y -444.174,Z 1377.690,A 0.000,B 0.000,C 90.000,E1 160.115} C_DIS
LIN {X -0.023,Y -456.714,Z 1377.684,A 0.000,B 0.000,C 90.000,E1 159.156} C_DIS
LIN {X -0.020,Y -465.905,Z 1377.680,A 0.000,B 0.000,C 90.000,E1 158.411} C_DIS
LIN {X -0.210,Y -473.420,Z 1377.677,A 0.000,B 0.000,C 90.000,E1 157.794} C_DIS
LIN {X 0.100,Y -480.762,Z 1377.673,A 0.000,B 0.000,C 90.000,E1 157.102} C_DIS
LIN {X 0.040,Y -489.373,Z 1377.668,A 0.000,B 0.000,C 90.000,E1 156.305} C_DIS
LIN {X -0.208,Y -494.990,Z 1377.665,A 0.000,B 0.000,C 90.000,E1 155.793} C_DIS
LIN {X 0.146,Y -501.817,Z 1377.661,A 0.000,B 0.000,C 90.000,E1 155.049} C_DIS
LIN {X -0.196,Y -505.732,Z 1377.659,A 0.000,B 0.000,C 90.000,E1 154.665} C_DIS
LIN {X -0.065,Y -513.396,Z 1377.654,A 0.000,B 0.000,C 90.000,E1 153.768} C_DIS
LIN {X 0.245,Y -519.411,Z 1377.650,A 0.000,B 0.000,C 90.000,E1 152.999} C_DIS
LIN {X 0.047,Y -523.889,Z 1377.647,A 0.000,B 0.000,C 90.000,E1 152.436} C_DIS
LIN {X -0.189,Y -527.034,Z 1377.645,A 0.000,B 0.000,C 90.000,E1 152.025} C_DIS
LIN {X -0.087,Y -530.724,Z 1377.641,A 0.000,B 0.000,C 90.000,E1 151.435} C_DIS
LIN {X 0.043,Y -533.942,Z 1377.638,A 0.000,B 0.000,C 90.000,E1 150.845} C_DIS
LIN {X 0.057,Y -537.337,Z 1377.634,A 0.000,B 0.000,C 90.000,E1 150.127} C_DIS
LIN {X 0.095,Y -540.232,Z 1377.630,A 0.000,B 0.000,C 90.000,E1 149.410} C_DIS
LIN {X -0.176,Y -542.311,Z 1377.627,A 0.000,B 0.000,C 90.000,E1 148.869} C_DIS
LIN {X 0.031,Y -544.172,Z 1377.624,A 0.000,B 0.000,C 90.000,E1 148.280} C_DIS
LIN {X -0.186,Y -546.438,Z 1377.619,A 0.000,B 0.000,C 90.000,E1 147.454} C_DIS
LIN {X 0.084,Y -548.340,Z 1377.614,A 0.000,B 0.000,C 90.000,E1 146.580} C_DIS
LIN {X -0.087,Y -549.960,Z 1377.610,A 0.000,B 0.000,C 90.000,E1 145.754} C_DIS
LIN {X 0.017,Y -550.851,Z 1377.607,A 0.000,B 0.000,C 90.000,E1 145.182} C_DIS
LIN {X -0.067,Y -552.414,Z 1377.600,A 0.000,B 0.000,C 90.000,E1 144.069} C_DIS
LIN {X 0.192,Y -553.492,Z 1377.594,A 0.000,B 0.000,C 90.000,E1 142.924} C_DIS
LIN {X 0.030,Y -554.333,Z 1377.588,A 0.000,B 0.000,C 90.000,E1 141.823} C_DIS
LIN {X -0.046,Y -555.285,Z 1377.580,A 0.000,B 0.000,C 90.000,E1 140.436} C_DIS
LIN {X 0.245,Y -556.089,Z 1377.573,A 0.000,B 0.000,C 90.000,E1 139.013} C_DIS
LIN {X 0.129,Y -556.845,Z 1377.565,A 0.000,B 0.000,C 90.000,E1 137.634} C_DIS
LIN {X -0.001,Y -557.418,Z 1377.557,A 0.000,B 0.000,C 90.000,E1 136.257} C_DIS
LIN {X -0.050,Y -558.024,Z 1377.548,A 0.000,B 0.000,C 90.000,E1 134.595} C_DIS
LIN {X -0.157,Y -558.542,Z 1377.540,A 0.000,B 0.000,C 90.000,E1 133.218} C_DIS
LIN {X -0.233,Y -558.946,Z 1377.532,A 0.000,B 0.000,C 90.000,E1 131.838} C_DIS
LIN {X 0.041,Y -559.239,Z 1377.526,A 0.000,B 0.000,C 90.000,E1 130.701} C_DIS
LIN {X 0.152,Y -560.132,Z 1377.515,A 0.000,B 0.000,C 90.000,E1 128.749} C_DIS
LIN {X -0.230,Y -560.796,Z 1377.512,A 0.000,B 0.000,C 90.000,E1 128.096} C_DIS
LIN {X 0.178,Y -561.155,Z 1377.511,A 0.000,B 0.000,C 90.000,E1 127.890} C_DIS
LIN {X 0.136,Y -561.202,Z 1377.511,A 0.000,B 0.000,C 90.000,E1 127.890} C_DIS
LIN {X -0.135,Y -562.314,Z 1377.510,A 0.000,B 0.000,C 90.000,E1 127.810} C_DIS
LIN {X 0.085,Y -563.333,Z 1377.509,A 0.000,B 0.000,C 90.000,E1 127.649} C_DIS
LIN {X 0.027,Y -563.777,Z 1377.509,A 0.000,B 0.000,C 90.000,E1 127.569} C_DIS
LIN {X 0.187,Y -567.967,Z 1377.508,A 0.000,B 0.000,C 90.000,E1 127.363} C_DIS
LIN {X -0.116,Y -573.871,Z 1377.507,A 0.000,B 0.000,C 90.000,E1 127.237} C_DIS
LIN {X -0.025,Y -580.529,Z 1377.506,A 0.000,B 0.000,C 90.000,E1 127.030} C_DIS
LIN {X -0.155,Y -586.666,Z 1377.504,A 0.000,B 0.000,C 90.000,E1 126.790} C_DIS
LIN {X 0.128,Y -592.423,Z 1377.503,A 0.000,B 0.000,C 90.000,E1 126.457} C_DIS
LIN {X -0.082,Y -596.627,Z 1377.501,A 0.000,B 0.000,C 90.000,E1 126.217} C_DIS
LIN {X 0.049,Y -599.523,Z 1377.500,A 0.000,B 0.000,C 90.000,E1 126.011} C_DIS
LIN {X -0.105,Y -605.107,Z 1377.498,A 0.000,B 0.000,C 90.000,E1 125.598} C_DIS
LIN {X -0.295,Y -607.855,Z 1377.496,A 0.000,B 0.000,C 90.000,E1 125.391} C_DIS
LIN {X -0.159,Y -614.093,Z 1377.493,A 0.000,B 0.000,C 90.000,E1 124.818} C_DIS
LIN {X -0.055,Y -619.105,Z 1377.491,A 0.000,B 0.000,C 90.000,E1 124.326} C_DIS
LIN {X -0.018,Y -623.888,Z 1377.488,A 0.000,B 0.000,C 90.000,E1 123.833} C_DIS
LIN {X 0.324,Y -628.527,Z 1377.485,A 0.000,B 0.000,C 90.000,E1 123.293} C_DIS
LIN {X 0.158,Y -633.926,Z 1377.482,A 0.000,B 0.000,C 90.000,E1 122.673} C_DIS
LIN {X 0.029,Y -638.755,Z 1377.478,A 0.000,B 0.000,C 90.000,E1 122.054} C_DIS
LIN {X 0.121,Y -642.501,Z 1377.475,A 0.000,B 0.000,C 90.000,E1 121.544} C_DIS
LIN {X 0.027,Y -645.846,Z 1377.473,A 0.000,B 0.000,C 90.000,E1 121.052} C_DIS
LIN {X -0.342,Y -649.588,Z 1377.469,A 0.000,B 0.000,C 90.000,E1 120.463} C_DIS
LIN {X 0.163,Y -652.309,Z 1377.466,A 0.000,B 0.000,C 90.000,E1 119.922} C_DIS
LIN {X -0.157,Y -655.093,Z 1377.463,A 0.000,B 0.000,C 90.000,E1 119.333} C_DIS
LIN {X -0.048,Y -656.094,Z 1377.462,A 0.000,B 0.000,C 90.000,E1 119.077} C_DIS
LIN {X -0.280,Y -658.535,Z 1377.458,A 0.000,B 0.000,C 90.000,E1 118.359} C_DIS
LIN {X 0.095,Y -659.986,Z 1377.453,A 0.000,B 0.000,C 90.000,E1 117.590} C_DIS
LIN {X 0.225,Y -660.247,Z 1377.452,A 0.000,B 0.000,C 90.000,E1 117.334} C_DIS
LIN {X -0.099,Y -660.395,Z 1377.449,A 0.000,B 0.000,C 90.000,E1 116.873} C_DIS
LIN {X 0.297,Y -660.252,Z 1377.445,A 0.000,B 0.000,C 90.000,E1 116.104} C_DIS
LIN {X -0.034,Y -659.886,Z 1377.443,A 0.000,B 0.000,C 90.000,E1 115.643} C_DIS
LIN {X -0.059,Y -659.339,Z 1377.440,A 0.000,B 0.000,C 90.000,E1 115.155} C_DIS
LIN {X 0.197,Y -658.386,Z 1377.437,A 0.000,B 0.000,C 90.000,E1 114.643} C_DIS
LIN {X 0.322,Y -657.648,Z 1377.436,A 0.000,B 0.000,C 90.000,E1 114.387} C_DIS
LIN {X -0.307,Y -655.149,Z 1377.433,A 0.000,B 0.000,C 90.000,E1 113.951} C_DIS
LIN {X -0.250,Y -654.268,Z 1377.432,A 0.000,B 0.000,C 90.000,E1 113.823} C_DIS
LIN {X -0.255,Y -649.363,Z 1377.430,A 0.000,B 0.000,C 90.000,E1 113.334} C_DIS
LIN {X -0.164,Y -647.572,Z 1377.429,A 0.000,B 0.000,C 90.000,E1 113.206} C_DIS
LIN {X 0.169,Y -645.650,Z 1377.428,A 0.000,B 0.000,C 90.000,E1 113.078} C_DIS
LIN {X 0.289,Y -640.429,Z 1377.427,A 0.000,B 0.000,C 90.000,E1 112.823} C_DIS
LIN {X 0.001,Y -638.424,Z 1377.427,A 0.000,B 0.000,C 90.000,E1 112.770} C_DIS
LIN {X -0.087,Y -634.208,Z 1377.426,A 0.000,B 0.000,C 90.000,E1 112.642} C_DIS
LIN {X -0.026,Y -620.762,Z 1377.424,A 0.000,B 0.000,C 90.000,E1 112.280} C_DIS
LIN {X -0.090,Y -620.807,Z 1377.424,A 0.000,B 0.000,C 90.000,E1 112.280} C_DIS
LIN {X -0.226,Y -628.650,Z 1377.419,A 0.000,B 0.000,C 90.000,E1 111.461} C_DIS
LIN {X 0.164,Y -633.310,Z 1377.416,A 0.000,B 0.000,C 90.000,E1 110.918} C_DIS
LIN {X -0.010,Y -637.542,Z 1377.414,A 0.000,B 0.000,C 90.000,E1 110.429} C_DIS
LIN {X -0.138,Y -642.128,Z 1377.410,A 0.000,B 0.000,C 90.000,E1 109.812} C_DIS
LIN {X 0.375,Y -646.073,Z 1377.407,A 0.000,B 0.000,C 90.000,E1 109.141} C_DIS
LIN {X -0.040,Y -650.833,Z 1377.402,A 0.000,B 0.000,C 90.000,E1 108.308} C_DIS
LIN {X -0.071,Y -653.984,Z 1377.398,A 0.000,B 0.000,C 90.000,E1 107.692} C_DIS
LIN {X -0.321,Y -656.352,Z 1377.396,A 0.000,B 0.000,C 90.000,E1 107.221} C_DIS
LIN {X 0.269,Y -658.429,Z 1377.393,A 0.000,B 0.000,C 90.000,E1 106.677} C_DIS
LIN {X 0.159,Y -659.414,Z 1377.391,A 0.000,B 0.000,C 90.000,E1 106.441} C_DIS
LIN {X 0.031,Y -661.729,Z 1377.387,A 0.000,B 0.000,C 90.000,E1 105.717} C_DIS
LIN {X -0.256,Y -663.383,Z 1377.383,A 0.000,B 0.000,C 90.000,E1 105.009} C_DIS
LIN {X 0.205,Y -664.287,Z 1377.381,A 0.000,B 0.000,C 90.000,E1 104.481} C_DIS
LIN {X -0.051,Y -665.210,Z 1377.377,A 0.000,B 0.000,C 90.000,E1 103.772} C_DIS
LIN {X -0.218,Y -665.642,Z 1377.374,A 0.000,B 0.000,C 90.000,E1 103.300} C_DIS
LIN {X 0.267,Y -665.842,Z 1377.371,A 0.000,B 0.000,C 90.000,E1 102.771} C_DIS
LIN {X 0.021,Y -665.746,Z 1377.367,A 0.000,B 0.000,C 90.000,E1 102.063} C_DIS
LIN {X -0.147,Y -665.479,Z 1377.364,A 0.000,B 0.000,C 90.000,E1 101.591} C_DIS
LIN {X 0.204,Y -664.963,Z 1377.362,A 0.000,B 0.000,C 90.000,E1 101.074} C_DIS
LIN {X 0.029,Y -664.234,Z 1377.359,A 0.000,B 0.000,C 90.000,E1 100.602} C_DIS
LIN {X 0.288,Y -662.773,Z 1377.355,A 0.000,B 0.000,C 90.000,E1 99.849} C_DIS
LIN {X 0.092,Y -661.573,Z 1377.352,A 0.000,B 0.000,C 90.000,E1 99.378} C_DIS
LIN {X -0.221,Y -660.090,Z 1377.349,A 0.000,B 0.000,C 90.000,E1 98.916} C_DIS
LIN {X -0.003,Y -657.495,Z 1377.345,A 0.000,B 0.000,C 90.000,E1 98.163} C_DIS
LIN {X 0.314,Y -655.561,Z 1377.343,A 0.000,B 0.000,C 90.000,E1 97.644} C_DIS
LIN {X -0.029,Y -653.392,Z 1377.340,A 0.000,B 0.000,C 90.000,E1 97.182} C_DIS
LIN {X 0.117,Y -649.651,Z 1377.336,A 0.000,B 0.000,C 90.000,E1 96.429} C_DIS
LIN {X -0.221,Y -647.625,Z 1377.334,A 0.000,B 0.000,C 90.000,E1 96.087} C_DIS
LIN {X 0.255,Y -641.660,Z 1377.328,A 0.000,B 0.000,C 90.000,E1 95.049} C_DIS
LIN {X -0.179,Y -638.522,Z 1377.325,A 0.000,B 0.000,C 90.000,E1 94.588} C_DIS
LIN {X -0.128,Y -634.123,Z 1377.322,A 0.000,B 0.000,C 90.000,E1 93.955} C_DIS
LIN {X -0.021,Y -630.199,Z 1377.319,A 0.000,B 0.000,C 90.000,E1 93.440} C_DIS
LIN {X -0.045,Y -624.387,Z 1377.316,A 0.000,B 0.000,C 90.000,E1 92.808} C_DIS
LIN {X 0.051,Y -617.985,Z 1377.312,A 0.000,B 0.000,C 90.000,E1 92.178} C_DIS
LIN {X 0.284,Y -610.127,Z 1377.308,A 0.000,B 0.000,C 90.000,E1 91.432} C_DIS
LIN {X 0.137,Y -604.449,Z 1377.306,A 0.000,B 0.000,C 90.000,E1 90.974} C_DIS
LIN {X 0.165,Y -603.039,Z 1377.305,A 0.000,B 0.000,C 90.000,E1 90.859} C_DIS
LIN {X 0.040,Y -596.805,Z 1377.303,A 0.000,B 0.000,C 90.000,E1 90.458} C_DIS
LIN {X -0.165,Y -593.301,Z 1377.302,A 0.000,B 0.000,C 90.000,E1 90.286} C_DIS
LIN {X 0.112,Y -588.172,Z 1377.300,A 0.000,B 0.000,C 90.000,E1 90.000} C_DIS
LIN {X 0.135,Y -578.358,Z 1377.298,A 0.000,B 0.000,C 90.000,E1 89.542} C_DIS
LIN {X -0.092,Y -576.981,Z 1377.297,A 0.000,B 0.000,C 90.000,E1 89.484} C_DIS
LIN {X 0.258,Y -575.962,Z 1377.297,A 0.000,B 0.000,C 90.000,E1 89.370} C_DIS
LIN {X -0.123,Y -574.061,Z 1377.296,A 0.000,B 0.000,C 90.000,E1 89.198} C_DIS
LIN {X 0.105,Y -573.770,Z 1377.295,A 0.000,B 0.000,C 90.000,E1 89.026} C_DIS
LIN {X 0.249,Y -573.630,Z 1377.293,A 0.000,B 0.000,C 90.000,E1 88.740} C_DIS
LIN {X 0.121,Y -574.090,Z 1377.289,A 0.000,B 0.000,C 90.000,E1 87.993} C_DIS
LIN {X 0.195,Y -575.946,Z 1377.277,A 0.000,B 0.000,C 90.000,E1 85.812} C_DIS
LIN {X -0.221,Y -578.167,Z 1377.265,A 0.000,B 0.000,C 90.000,E1 83.685} C_DIS
LIN {X 0.119,Y -579.765,Z 1377.257,A 0.000,B 0.000,C 90.000,E1 82.299} C_DIS
LIN {X -0.091,Y -581.384,Z 1377.250,A 0.000,B 0.000,C 90.000,E1 80.971} C_DIS
LIN {X 0.049,Y -583.290,Z 1377.241,A 0.000,B 0.000,C 90.000,E1 79.342} C_DIS
LIN {X 0.100,Y -584.679,Z 1377.233,A 0.000,B 0.000,C 90.000,E1 77.993} C_DIS
LIN {X -0.147,Y -586.103,Z 1377.224,A 0.000,B 0.000,C 90.000,E1 76.408} C_DIS
LIN {X -0.228,Y -587.301,Z 1377.216,A 0.000,B 0.000,C 90.000,E1 74.810} C_DIS
LIN {X 0.025,Y -588.149,Z 1377.208,A 0.000,B 0.000,C 90.000,E1 73.449} C_DIS
LIN {X 0.313,Y -589.110,Z 1377.199,A 0.000,B 0.000,C 90.000,E1 71.819} C_DIS
LIN {X -0.254,Y -590.175,Z 1377.189,A 0.000,B 0.000,C 90.000,E1 70.007} C_DIS
LIN {X -0.061,Y -591.576,Z 1377.176,A 0.000,B 0.000,C 90.000,E1 67.592} C_DIS
LIN {X 0.178,Y -593.433,Z 1377.162,A 0.000,B 0.000,C 90.000,E1 65.177} C_DIS
LIN {X -0.295,Y -594.492,Z 1377.155,A 0.000,B 0.000,C 90.000,E1 63.896} C_DIS
LIN {X 0.056,Y -595.482,Z 1377.147,A 0.000,B 0.000,C 90.000,E1 62.538} C_DIS
LIN {X 0.376,Y -597.564,Z 1377.134,A 0.000,B 0.000,C 90.000,E1 60.127} C_DIS
LIN {X -0.041,Y -599.059,Z 1377.125,A 0.000,B 0.000,C 90.000,E1 58.584} C_DIS
LIN {X 0.073,Y -600.540,Z 1377.117,A 0.000,B 0.000,C 90.000,E1 56.993} C_DIS
LIN {X -0.129,Y -601.530,Z 1377.111,A 0.000,B 0.000,C 90.000,E1 55.960} C_DIS
LIN {X -0.055,Y -603.171,Z 1377.101,A 0.000,B 0.000,C 90.000,E1 54.116} C_DIS
LIN {X -0.197,Y -604.613,Z 1377.092,A 0.000,B 0.000,C 90.000,E1 52.557} C_DIS
LIN {X -0.213,Y -605.598,Z 1377.085,A 0.000,B 0.000,C 90.000,E1 51.251} C_DIS
LIN {X -0.097,Y -606.142,Z 1377.079,A 0.000,B 0.000,C 90.000,E1 50.194} C_DIS
LIN {X 0.295,Y -606.752,Z 1377.072,A 0.000,B 0.000,C 90.000,E1 48.852} C_DIS
LIN {X -0.024,Y -607.110,Z 1377.066,A 0.000,B 0.000,C 90.000,E1 47.838} C_DIS
LIN {X 0.107,Y -607.317,Z 1377.060,A 0.000,B 0.000,C 90.000,E1 46.782} C_DIS
LIN {X -0.163,Y -607.383,Z 1377.051,A 0.000,B 0.000,C 90.000,E1 45.243} C_DIS
LIN {X -0.241,Y -607.084,Z 1377.044,A 0.000,B 0.000,C 90.000,E1 43.947} C_DIS
LIN {X 0.048,Y -606.799,Z 1377.040,A 0.000,B 0.000,C 90.000,E1 43.137} C_DIS
LIN {X -0.020,Y -606.170,Z 1377.032,A 0.000,B 0.000,C 90.000,E1 41.838} C_DIS
LIN {X 0.106,Y -605.595,Z 1377.027,A 0.000,B 0.000,C 90.000,E1 40.782} C_DIS
LIN {X 0.224,Y -604.912,Z 1377.021,A 0.000,B 0.000,C 90.000,E1 39.725} C_DIS
LIN {X -0.264,Y -603.833,Z 1377.014,A 0.000,B 0.000,C 90.000,E1 38.463} C_DIS
LIN {X 0.291,Y -602.830,Z 1377.008,A 0.000,B 0.000,C 90.000,E1 37.363} C_DIS
LIN {X -0.023,Y -601.580,Z 1377.002,A 0.000,B 0.000,C 90.000,E1 36.343} C_DIS
LIN {X 0.370,Y -600.427,Z 1376.998,A 0.000,B 0.000,C 90.000,E1 35.518} C_DIS
LIN {X 0.264,Y -598.994,Z 1376.993,A 0.000,B 0.000,C 90.000,E1 34.739} C_DIS
LIN {X -0.064,Y -596.115,Z 1376.986,A 0.000,B 0.000,C 90.000,E1 33.452} C_DIS
LIN {X 0.061,Y -594.878,Z 1376.983,A 0.000,B 0.000,C 90.000,E1 32.911} C_DIS
LIN {X -0.111,Y -592.771,Z 1376.979,A 0.000,B 0.000,C 90.000,E1 32.133} C_DIS
LIN {X 0.075,Y -589.614,Z 1376.973,A 0.000,B 0.000,C 90.000,E1 31.052} C_DIS
LIN {X 0.033,Y -586.729,Z 1376.968,A 0.000,B 0.000,C 90.000,E1 30.256} C_DIS
LIN {X -0.040,Y -583.550,Z 1376.964,A 0.000,B 0.000,C 90.000,E1 29.461} C_DIS
LIN {X 0.362,Y -579.967,Z 1376.959,A 0.000,B 0.000,C 90.000,E1 28.615} C_DIS
LIN {X 0.012,Y -576.715,Z 1376.955,A 0.000,B 0.000,C 90.000,E1 27.975} C_DIS
LIN {X 0.254,Y -571.727,Z 1376.950,A 0.000,B 0.000,C 90.000,E1 27.001} C_DIS
LIN {X 0.173,Y -566.165,Z 1376.945,A 0.000,B 0.000,C 90.000,E1 26.052} C_DIS
LIN {X 0.270,Y -560.130,Z 1376.940,A 0.000,B 0.000,C 90.000,E1 25.079} C_DIS
LIN {X -0.035,Y -557.329,Z 1376.937,A 0.000,B 0.000,C 90.000,E1 24.695} C_DIS
LIN {X 0.325,Y -551.341,Z 1376.933,A 0.000,B 0.000,C 90.000,E1 23.823} C_DIS
LIN {X 0.024,Y -545.943,Z 1376.929,A 0.000,B 0.000,C 90.000,E1 23.153} C_DIS
LIN {X -0.106,Y -540.111,Z 1376.925,A 0.000,B 0.000,C 90.000,E1 22.461} C_DIS
LIN {X 0.128,Y -532.884,Z 1376.920,A 0.000,B 0.000,C 90.000,E1 21.589} C_DIS
LIN {X 0.064,Y -522.567,Z 1376.914,A 0.000,B 0.000,C 90.000,E1 20.482} C_DIS
LIN {X 0.125,Y -513.411,Z 1376.908,A 0.000,B 0.000,C 90.000,E1 19.504} C_DIS
LIN {X -0.197,Y -502.387,Z 1376.902,A 0.000,B 0.000,C 90.000,E1 18.417} C_DIS
LIN {X 0.239,Y -491.612,Z 1376.896,A 0.000,B 0.000,C 90.000,E1 17.275} C_DIS
LIN {X 0.122,Y -479.030,Z 1376.889,A 0.000,B 0.000,C 90.000,E1 16.024} C_DIS
LIN {X -0.186,Y -466.397,Z 1376.882,A 0.000,B 0.000,C 90.000,E1 14.773} C_DIS
LIN {X 0.017,Y -455.010,Z 1376.876,A 0.000,B 0.000,C 90.000,E1 13.592} C_DIS
LIN {X 0.035,Y -438.238,Z 1376.866,A 0.000,B 0.000,C 90.000,E1 11.827} C_DIS
LIN {X 0.009,Y -421.596,Z 1376.855,A 0.000,B 0.000,C 90.000,E1 9.962} C_DIS
LIN {X 0.174,Y -410.484,Z 1376.848,A 0.000,B 0.000,C 90.000,E1 8.624} C_DIS
LIN {X -0.145,Y -400.757,Z 1376.842,A 0.000,B 0.000,C 90.000,E1 7.530} C_DIS
LIN {X 0.069,Y -396.614,Z 1376.839,A 0.000,B 0.000,C 90.000,E1 7.004} C_DIS
LIN {X 0.195,Y -392.208,Z 1376.836,A 0.000,B 0.000,C 90.000,E1 6.372} C_DIS
LIN {X -0.163,Y -391.456,Z 1376.835,A 0.000,B 0.000,C 90.000,E1 6.258} C_DIS
LIN {X 0.188,Y -391.449,Z 1376.835,A 0.000,B 0.000,C 90.000,E1 6.201} C_DIS
LIN {X -0.009,Y -394.254,Z 1376.833,A 0.000,B 0.000,C 90.000,E1 5.853} C_DIS
LIN {X -0.004,Y -399.553,Z 1376.830,A 0.000,B 0.000,C 90.000,E1 5.391} C_DIS
LIN {X 0.082,Y -405.455,Z 1376.828,A 0.000,B 0.000,C 90.000,E1 4.935} C_DIS
LIN {X -0.134,Y -410.246,Z 1376.825,A 0.000,B 0.000,C 90.000,E1 4.588} C_DIS
LIN {X -0.158,Y -417.525,Z 1376.822,A 0.000,B 0.000,C 90.000,E1 3.898} C_DIS
LIN {X 0.161,Y -424.353,Z 1376.817,A 0.000,B 0.000,C 90.000,E1 3.094} C_DIS
LIN {X -0.040,Y -430.847,Z 1376.813,A 0.000,B 0.000,C 90.000,E1 2.293} C_DIS
LIN {X 0.222,Y -438.120,Z 1376.807,A 0.000,B 0.000,C 90.000,E1 1.260} C_DIS
LIN {X -0.058,Y -441.661,Z 1376.804,A 0.000,B 0.000,C 90.000,E1 0.802} C_DIS
LIN {X 0.000,Y -447.097,Z 1376.800,A 0.000,B 0.000,C 90.000,E1 360.000} C_DIS
LIN {X 0.024,Y -452.576,Z 1376.795,A 0.000,B 0.000,C 90.000,E1 359.141} C_DIS
LIN {X -0.002,Y -457.452,Z 1376.791,A 0.000,B 0.000,C 90.000,E1 358.339} C_DIS
LIN {X -0.068,Y -461.085,Z 1376.787,A 0.000,B 0.000,C 90.000,E1 357.707} C_DIS
LIN {X 0.114,Y -466.107,Z 1376.782,A 0.000,B 0.000,C 90.000,E1 356.731} C_DIS
LIN {X 0.094,Y -469.237,Z 1376.778,A 0.000,B 0.000,C 90.000,E1 356.102} C_DIS
LIN {X -0.064,Y -473.476,Z 1376.773,A 0.000,B 0.000,C 90.000,E1 355.179} C_DIS
LIN {X 0.134,Y -476.719,Z 1376.769,A 0.000,B 0.000,C 90.000,E1 354.375} C_DIS
LIN {X 0.227,Y -479.151,Z 1376.765,A 0.000,B 0.000,C 90.000,E1 353.742} C_DIS
LIN {X 0.183,Y -482.514,Z 1376.760,A 0.000,B 0.000,C 90.000,E1 352.818} C_DIS
LIN {X -0.167,Y -484.563,Z 1376.757,A 0.000,B 0.000,C 90.000,E1 352.243} C_DIS
LIN {X -0.082,Y -487.353,Z 1376.752,A 0.000,B 0.000,C 90.000,E1 351.310} C_DIS
LIN {X -0.037,Y -489.843,Z 1376.747,A 0.000,B 0.000,C 90.000,E1 350.387} C_DIS
LIN {X 0.115,Y -492.069,Z 1376.742,A 0.000,B 0.000,C 90.000,E1 349.454} C_DIS
LIN {X 0.011,Y -492.686,Z 1376.740,A 0.000,B 0.000,C 90.000,E1 349.162} C_DIS
LIN {X -0.091,Y -493.135,Z 1376.738,A 0.000,B 0.000,C 90.000,E1 348.870} C_DIS
LIN {X -0.191,Y -493.390,Z 1376.736,A 0.000,B 0.000,C 90.000,E1 348.578} C_DIS
LIN {X 0.195,Y -493.395,Z 1376.735,A 0.000,B 0.000,C 90.000,E1 348.229} C_DIS
LIN {X 0.097,Y -492.938,Z 1376.733,A 0.000,B 0.000,C 90.000,E1 347.937} C_DIS
LIN {X -0.140,Y -492.368,Z 1376.732,A 0.000,B 0.000,C 90.000,E1 347.813} C_DIS
LIN {X 0.000,Y -491.055,Z 1376.731,A 0.000,B 0.000,C 90.000,E1 347.645} C_DIS
LIN {X -0.102,Y -481.850,Z 1376.730,A 0.000,B 0.000,C 90.000,E1 347.409} C_DIS
LIN {X -0.141,Y -444.379,Z 1376.724,A 0.000,B 0.000,C 90.000,E1 346.353} C_DIS
LIN {X 0.014,Y -412.707,Z 1376.718,A 0.000,B 0.000,C 90.000,E1 345.283} C_DIS
LIN {X -0.009,Y -384.721,Z 1376.712,A 0.000,B 0.000,C 90.000,E1 344.212} C_DIS
LIN {X -0.177,Y -359.844,Z 1376.706,A 0.000,B 0.000,C 90.000,E1 343.142} C_DIS
LIN {X 0.134,Y -359.843,Z 1376.706,A 0.000,B 0.000,C 90.000,E1 343.087} C_DIS
LIN {X 0.015,Y -361.972,Z 1376.682,A 0.000,B 0.000,C 90.000,E1 338.847} C_DIS
LIN {X -0.066,Y -365.894,Z 1376.643,A 0.000,B 0.000,C 90.000,E1 331.769} C_DIS
LIN {X 0.013,Y -366.206,Z 1376.641,A 0.000,B 0.000,C 90.000,E1 331.385} C_DIS
LIN {X 0.232,Y -371.254,Z 1376.604,A 0.000,B 0.000,C 90.000,E1 324.689} C_DIS
LIN {X 0.003,Y -371.687,Z 1376.602,A 0.000,B 0.000,C 90.000,E1 324.356} C_DIS
LIN {X -0.231,Y -377.247,Z 1376.567,A 0.000,B 0.000,C 90.000,E1 318.162} C_DIS
LIN {X 0.047,Y -378.177,Z 1376.563,A 0.000,B 0.000,C 90.000,E1 317.391} C_DIS
LIN {X 0.032,Y -383.825,Z 1376.531,A 0.000,B 0.000,C 90.000,E1 311.595} C_DIS
LIN {X 0.117,Y -384.813,Z 1376.527,A 0.000,B 0.000,C 90.000,E1 310.862} C_DIS
LIN {X -0.184,Y -390.986,Z 1376.493,A 0.000,B 0.000,C 90.000,E1 304.818} C_DIS
LIN {X 0.206,Y -391.380,Z 1376.491,A 0.000,B 0.000,C 90.000,E1 304.405} C_DIS
LIN {X 0.151,Y -396.716,Z 1376.460,A 0.000,B 0.000,C 90.000,E1 298.743} C_DIS
LIN {X 0.020,Y -397.084,Z 1376.458,A 0.000,B 0.000,C 90.000,E1 298.409} C_DIS
LIN {X 0.157,Y -401.512,Z 1376.427,A 0.000,B 0.000,C 90.000,E1 292.770} C_DIS
LIN {X 0.103,Y -401.773,Z 1376.423,A 0.000,B 0.000,C 90.000,E1 292.078} C_DIS
LIN {X -0.089,Y -404.585,Z 1376.396,A 0.000,B 0.000,C 90.000,E1 287.221} C_DIS
LIN {X 0.013,Y -404.758,Z 1376.394,A 0.000,B 0.000,C 90.000,E1 286.858} C_DIS
LIN {X -0.080,Y -406.052,Z 1376.365,A 0.000,B 0.000,C 90.000,E1 281.658} C_DIS
LIN {X 0.010,Y -406.128,Z 1376.363,A 0.000,B 0.000,C 90.000,E1 281.299} C_DIS
LIN {X 0.040,Y -405.660,Z 1376.334,A 0.000,B 0.000,C 90.000,E1 276.087} C_DIS
LIN {X 0.044,Y -405.585,Z 1376.332,A 0.000,B 0.000,C 90.000,E1 275.739} C_DIS
LIN {X 0.118,Y -403.542,Z 1376.305,A 0.000,B 0.000,C 90.000,E1 270.859} C_DIS
LIN {X 0.053,Y -403.016,Z 1376.301,A 0.000,B 0.000,C 90.000,E1 270.172} C_DIS
LIN {X -0.124,Y -398.998,Z 1376.272,A 0.000,B 0.000,C 90.000,E1 264.951} C_DIS
LIN {X 0.037,Y -392.906,Z 1376.241,A 0.000,B 0.000,C 90.000,E1 259.285} C_DIS
LIN {X 0.028,Y -391.832,Z 1376.237,A 0.000,B 0.000,C 90.000,E1 258.578} C_DIS
LIN {X 0.154,Y -385.708,Z 1376.211,A 0.000,B 0.000,C 90.000,E1 253.921} C_DIS
LIN {X 0.199,Y -384.926,Z 1376.207,A 0.000,B 0.000,C 90.000,E1 253.196} C_DIS
LIN {X -0.053,Y -378.083,Z 1376.183,A 0.000,B 0.000,C 90.000,E1 248.901} C_DIS
LIN {X 0.175,Y -376.329,Z 1376.175,A 0.000,B 0.000,C 90.000,E1 247.411} C_DIS
LIN {X 0.155,Y -375.807,Z 1376.173,A 0.000,B 0.000,C 90.000,E1 247.050} C_DIS
LIN {X -0.072,Y -369.050,Z 1376.150,A 0.000,B 0.000,C 90.000,E1 243.050} C_DIS
LIN {X 0.160,Y -366.200,Z 1376.138,A 0.000,B 0.000,C 90.000,E1 240.795} C_DIS
LIN {X 0.002,Y -358.798,Z 1376.113,A 0.000,B 0.000,C 90.000,E1 236.342} C_DIS
LIN {X 0.080,Y -355.988,Z 1376.100,A 0.000,B 0.000,C 90.000,E1 234.069} C_DIS
LIN {X -0.113,Y -348.910,Z 1376.075,A 0.000,B 0.000,C 90.000,E1 229.542} C_DIS
LIN {X 0.088,Y -345.833,Z 1376.060,A 0.000,B 0.000,C 90.000,E1 226.824} C_DIS
LIN {X -0.180,Y -339.080,Z 1376.032,A 0.000,B 0.000,C 90.000,E1 221.838} C_DIS
LIN {X -0.096,Y -336.924,Z 1376.019,A 0.000,B 0.000,C 90.000,E1 219.483} C_DIS
LIN {X 0.178,Y -331.258,Z 1375.991,A 0.000,B 0.000,C 90.000,E1 214.326} C_DIS
LIN {X -0.044,Y -329.347,Z 1375.975,A 0.000,B 0.000,C 90.000,E1 211.592} C_DIS
LIN {X 0.056,Y -328.204,Z 1375.969,A 0.000,B 0.000,C 90.000,E1 210.384} C_DIS
LIN {X 0.084,Y -323.961,Z 1375.931,A 0.000,B 0.000,C 90.000,E1 203.590} C_DIS
LIN {X -0.110,Y -323.639,Z 1375.927,A 0.000,B 0.000,C 90.000,E1 202.823} C_DIS
LIN {X -0.112,Y -321.757,Z 1375.908,A 0.000,B 0.000,C 90.000,E1 199.396} C_DIS
LIN {X -0.129,Y -321.809,Z 1375.908,A 0.000,B 0.000,C 90.000,E1 199.396} C_DIS
LIN {X -0.089,Y -344.424,Z 1375.901,A 0.000,B 0.000,C 90.000,E1 198.109} C_DIS
LIN {X 0.054,Y -369.426,Z 1375.894,A 0.000,B 0.000,C 90.000,E1 196.858} C_DIS
LIN {X 0.021,Y -396.367,Z 1375.887,A 0.000,B 0.000,C 90.000,E1 195.717} C_DIS
LIN {X -0.058,Y -425.255,Z 1375.881,A 0.000,B 0.000,C 90.000,E1 194.662} C_DIS
LIN {X -0.030,Y -439.787,Z 1375.879,A 0.000,B 0.000,C 90.000,E1 194.175} C_DIS
LIN {X -0.067,Y -442.466,Z 1375.878,A 0.000,B 0.000,C 90.000,E1 194.064} C_DIS
LIN {X 0.160,Y -443.610,Z 1375.877,A 0.000,B 0.000,C 90.000,E1 193.883} C_DIS
LIN {X -0.246,Y -444.361,Z 1375.876,A 0.000,B 0.000,C 90.000,E1 193.772} C_DIS
LIN {X -0.116,Y -444.902,Z 1375.875,A 0.000,B 0.000,C 90.000,E1 193.592} C_DIS
LIN {X 0.050,Y -445.605,Z 1375.874,A 0.000,B 0.000,C 90.000,E1 193.244} C_DIS
LIN {X -0.115,Y -446.021,Z 1375.872,A 0.000,B 0.000,C 90.000,E1 192.939} C_DIS
LIN {X -0.203,Y -446.317,Z 1375.868,A 0.000,B 0.000,C 90.000,E1 192.299} C_DIS
LIN {X 0.153,Y -446.506,Z 1375.865,A 0.000,B 0.000,C 90.000,E1 191.602} C_DIS
LIN {X 0.082,Y -446.650,Z 1375.857,A 0.000,B 0.000,C 90.000,E1 190.310} C_DIS
LIN {X -0.075,Y -446.645,Z 1375.850,A 0.000,B 0.000,C 90.000,E1 189.029} C_DIS
LIN {X -0.002,Y -446.569,Z 1375.839,A 0.000,B 0.000,C 90.000,E1 187.068} C_DIS
LIN {X 0.214,Y -446.509,Z 1375.832,A 0.000,B 0.000,C 90.000,E1 185.739} C_DIS
LIN {X -0.065,Y -446.269,Z 1375.825,A 0.000,B 0.000,C 90.000,E1 184.473} C_DIS
LIN {X -0.070,Y -445.783,Z 1375.819,A 0.000,B 0.000,C 90.000,E1 183.498} C_DIS
LIN {X -0.216,Y -445.374,Z 1375.816,A 0.000,B 0.000,C 90.000,E1 182.865} C_DIS
LIN {X 0.194,Y -444.368,Z 1375.810,A 0.000,B 0.000,C 90.000,E1 181.835} C_DIS
LIN {X 0.031,Y -443.592,Z 1375.807,A 0.000,B 0.000,C 90.000,E1 181.203} C_DIS
LIN {X -0.019,Y -442.113,Z 1375.801,A 0.000,B 0.000,C 90.000,E1 180.229} C_DIS
LIN {X -0.209,Y -440.957,Z 1375.798,A 0.000,B 0.000,C 90.000,E1 179.599} C_DIS
LIN {X 0.033,Y -439.615,Z 1375.794,A 0.000,B 0.000,C 90.000,E1 178.912} C_DIS
LIN {X -0.053,Y -437.123,Z 1375.789,A 0.000,B 0.000,C 90.000,E1 177.936} C_DIS
LIN {X -0.184,Y -433.839,Z 1375.783,A 0.000,B 0.000,C 90.000,E1 176.963} C_DIS
LIN {X 0.052,Y -430.638,Z 1375.778,A 0.000,B 0.000,C 90.000,E1 176.102} C_DIS
LIN {X -0.174,Y -426.875,Z 1375.774,A 0.000,B 0.000,C 90.000,E1 175.298} C_DIS
LIN {X 0.026,Y -422.310,Z 1375.769,A 0.000,B 0.000,C 90.000,E1 174.432} C_DIS
LIN {X 0.188,Y -415.934,Z 1375.764,A 0.000,B 0.000,C 90.000,E1 173.394} C_DIS
LIN {X -0.149,Y -407.852,Z 1375.757,A 0.000,B 0.000,C 90.000,E1 172.243} C_DIS
LIN {X -0.144,Y -394.375,Z 1375.745,A 0.000,B 0.000,C 90.000,E1 170.151} C_DIS
LIN {X 0.074,Y -384.112,Z 1375.735,A 0.000,B 0.000,C 90.000,E1 168.342} C_DIS
LIN {X 0.000,Y -382.341,Z 1375.733,A 0.000,B 0.000,C 90.000,E1 167.993} C_DIS
LIN {X 0.007,Y -379.407,Z 1375.729,A 0.000,B 0.000,C 90.000,E1 167.297} C_DIS
LIN {X -0.124,Y -378.044,Z 1375.726,A 0.000,B 0.000,C 90.000,E1 166.645} C_DIS
LIN {X 0.168,Y -378.012,Z 1375.725,A 0.000,B 0.000,C 90.000,E1 166.464} C_DIS
LIN {X 0.124,Y -381.395,Z 1375.722,A 0.000,B 0.000,C 90.000,E1 165.880} C_DIS
LIN {X 0.126,Y -386.608,Z 1375.718,A 0.000,B 0.000,C 90.000,E1 165.227} C_DIS
LIN {X -0.135,Y -392.249,Z 1375.715,A 0.000,B 0.000,C 90.000,E1 164.629} C_DIS
LIN {X -0.137,Y -400.556,Z 1375.710,A 0.000,B 0.000,C 90.000,E1 163.795} C_DIS
LIN {X -0.094,Y -417.697,Z 1375.701,A 0.000,B 0.000,C 90.000,E1 162.236} C_DIS
LIN {X 0.009,Y -443.121,Z 1375.690,A 0.000,B 0.000,C 90.000,E1 160.188} C_DIS
LIN {X 0.202,Y -455.564,Z 1375.685,A 0.000,B 0.000,C 90.000,E1 159.209} C_DIS
LIN {X 0.249,Y -464.798,Z 1375.681,A 0.000,B 0.000,C 90.000,E1 158.465} C_DIS
LIN {X 0.122,Y -472.267,Z 1375.677,A 0.000,B 0.000,C 90.000,E1 157.847} C_DIS
LIN {X -0.147,Y -478.191,Z 1375.674,A 0.000,B 0.000,C 90.000,E1 157.358} C_DIS
LIN {X 0.052,Y -485.479,Z 1375.670,A 0.000,B 0.000,C 90.000,E1 156.666} C_DIS
LIN {X -0.078,Y -494.067,Z 1375.666,A 0.000,B 0.000,C 90.000,E1 155.869} C_DIS
LIN {X -0.004,Y -502.171,Z 1375.661,A 0.000,B 0.000,C 90.000,E1 155.025} C_DIS
LIN {X 0.120,Y -506.048,Z 1375.659,A 0.000,B 0.000,C 90.000,E1 154.588} C_DIS
LIN {X 0.043,Y -513.686,Z 1375.654,A 0.000,B 0.000,C 90.000,E1 153.717} C_DIS
LIN {X 0.038,Y -518.553,Z 1375.651,A 0.000,B 0.000,C 90.000,E1 153.127} C_DIS
LIN {X 0.074,Y -523.086,Z 1375.648,A 0.000,B 0.000,C 90.000,E1 152.538} C_DIS
LIN {X 0.060,Y -526.301,Z 1375.645,A 0.000,B 0.000,C 90.000,E1 152.103} C_DIS
LIN {X 0.154,Y -530.060,Z 1375.642,A 0.000,B 0.000,C 90.000,E1 151.513} C_DIS
LIN {X 0.132,Y -534.106,Z 1375.638,A 0.000,B 0.000,C 90.000,E1 150.795} C_DIS
LIN {X 0.144,Y -537.472,Z 1375.634,A 0.000,B 0.000,C 90.000,E1 150.078} C_DIS
LIN {X -0.285,Y -540.313,Z 1375.630,A 0.000,B 0.000,C 90.000,E1 149.410} C_DIS
LIN {X 0.189,Y -542.378,Z 1375.627,A 0.000,B 0.000,C 90.000,E1 148.791} C_DIS
LIN {X -0.064,Y -544.204,Z 1375.624,A 0.000,B 0.000,C 90.000,E1 148.250} C_DIS
LIN {X 0.187,Y -546.434,Z 1375.619,A 0.000,B 0.000,C 90.000,E1 147.375} C_DIS
LIN {X 0.003,Y -548.297,Z 1375.614,A 0.000,B 0.000,C 90.000,E1 146.548} C_DIS
LIN {X -0.162,Y -549.862,Z 1375.609,A 0.000,B 0.000,C 90.000,E1 145.722} C_DIS
LIN {X 0.138,Y -551.184,Z 1375.605,A 0.000,B 0.000,C 90.000,E1 144.848} C_DIS
LIN {X -0.131,Y -552.330,Z 1375.600,A 0.000,B 0.000,C 90.000,E1 144.036} C_DIS
LIN {X -0.199,Y -553.377,Z 1375.594,A 0.000,B 0.000,C 90.000,E1 142.924} C_DIS
LIN {X 0.072,Y -554.207,Z 1375.588,A 0.000,B 0.000,C 90.000,E1 141.778} C_DIS
LIN {X -0.083,Y -554.980,Z 1375.582,A 0.000,B 0.000,C 90.000,E1 140.678} C_DIS
LIN {X -0.224,Y -555.825,Z 1375.574,A 0.000,B 0.000,C 90.000,E1 139.299} C_DIS
LIN {X -0.273,Y -556.718,Z 1375.565,A 0.000,B 0.000,C 90.000,E1 137.634} C_DIS
LIN {X -0.003,Y -557.296,Z 1375.557,A 0.000,B 0.000,C 90.000,E1 136.215} C_DIS
LIN {X -0.066,Y -557.903,Z 1375.547,A 0.000,B 0.000,C 90.000,E1 134.555} C_DIS
LIN {X -0.160,Y -558.420,Z 1375.540,A 0.000,B 0.000,C 90.000,E1 133.176} C_DIS
LIN {X 0.144,Y -558.865,Z 1375.532,A 0.000,B 0.000,C 90.000,E1 131.757} C_DIS
LIN {X -0.007,Y -559.870,Z 1375.518,A 0.000,B 0.000,C 90.000,E1 129.277} C_DIS
LIN {X -0.088,Y -561.132,Z 1375.513,A 0.000,B 0.000,C 90.000,E1 128.257} C_DIS
LIN {X 0.022,Y -561.531,Z 1375.512,A 0.000,B 0.000,C 90.000,E1 128.177} C_DIS
LIN {X 0.009,Y -563.882,Z 1375.511,A 0.000,B 0.000,C 90.000,E1 127.971} C_DIS
LIN {X 0.121,Y -564.991,Z 1375.511,A 0.000,B 0.000,C 90.000,E1 127.890} C_DIS
LIN {X -0.377,Y -568.954,Z 1375.510,A 0.000,B 0.000,C 90.000,E1 127.810} C_DIS
LIN {X -0.095,Y -576.888,Z 1375.509,A 0.000,B 0.000,C 90.000,E1 127.569} C_DIS
LIN {X -0.094,Y -583.187,Z 1375.508,A 0.000,B 0.000,C 90.000,E1 127.363} C_DIS
LIN {X 0.004,Y -588.863,Z 1375.506,A 0.000,B 0.000,C 90.000,E1 127.076} C_DIS
LIN {X -0.178,Y -594.916,Z 1375.504,A 0.000,B 0.000,C 90.000,E1 126.744} C_DIS
LIN {X -0.130,Y -599.141,Z 1375.503,A 0.000,B 0.000,C 90.000,E1 126.457} C_DIS
LIN {X 0.095,Y -604.754,Z 1375.500,A 0.000,B 0.000,C 90.000,E1 126.011} C_DIS
LIN {X -0.302,Y -610.203,Z 1375.498,A 0.000,B 0.000,C 90.000,E1 125.598} C_DIS
LIN {X -0.127,Y -615.319,Z 1375.495,A 0.000,B 0.000,C 90.000,E1 125.105} C_DIS
LIN {X -0.098,Y -620.280,Z 1375.492,A 0.000,B 0.000,C 90.000,E1 124.612} C_DIS
LIN {X -0.211,Y -626.318,Z 1375.489,A 0.000,B 0.000,C 90.000,E1 123.992} C_DIS
LIN {X 0.146,Y -630.779,Z 1375.486,A 0.000,B 0.000,C 90.000,E1 123.452} C_DIS
LIN {X 0.001,Y -636.046,Z 1375.482,A 0.000,B 0.000,C 90.000,E1 122.832} C_DIS
LIN {X -0.107,Y -640.819,Z 1375.479,A 0.000,B 0.000,C 90.000,E1 122.212} C_DIS
LIN {X 0.339,Y -644.395,Z 1375.476,A 0.000,B 0.000,C 90.000,E1 121.671} C_DIS
LIN {X -0.077,Y -647.702,Z 1375.473,A 0.000,B 0.000,C 90.000,E1 121.209} C_DIS
LIN {X -0.140,Y -650.711,Z 1375.471,A 0.000,B 0.000,C 90.000,E1 120.718} C_DIS
LIN {X 0.094,Y -654.004,Z 1375.467,A 0.000,B 0.000,C 90.000,E1 120.079} C_DIS
LIN {X 0.116,Y -656.780,Z 1375.464,A 0.000,B 0.000,C 90.000,E1 119.461} C_DIS
LIN {X -0.111,Y -659.379,Z 1375.460,A 0.000,B 0.000,C 90.000,E1 118.743} C_DIS
LIN {X 0.140,Y -660.682,Z 1375.457,A 0.000,B 0.000,C 90.000,E1 118.231} C_DIS
LIN {X -0.181,Y -661.672,Z 1375.454,A 0.000,B 0.000,C 90.000,E1 117.769} C_DIS
LIN {X -0.047,Y -661.975,Z 1375.453,A 0.000,B 0.000,C 90.000,E1 117.513} C_DIS
LIN {X -0.226,Y -662.207,Z 1375.449,A 0.000,B 0.000,C 90.000,E1 116.796} C_DIS
LIN {X 0.048,Y -662.112,Z 1375.446,A 0.000,B 0.000,C 90.000,E1 116.283} C_DIS
LIN {X 0.173,Y -661.559,Z 1375.442,A 0.000,B 0.000,C 90.000,E1 115.540} C_DIS
LIN {X -0.154,Y -661.012,Z 1375.439,A 0.000,B 0.000,C 90.000,E1 115.079} C_DIS
LIN {X -0.164,Y -659.976,Z 1375.437,A 0.000,B 0.000,C 90.000,E1 114.591} C_DIS
LIN {X -0.033,Y -659.159,Z 1375.435,A 0.000,B 0.000,C 90.000,E1 114.335} C_DIS
LIN {X 0.217,Y -656.557,Z 1375.432,A 0.000,B 0.000,C 90.000,E1 113.823} C_DIS
LIN {X 0.275,Y -655.590,Z 1375.432,A 0.000,B 0.000,C 90.000,E1 113.695} C_DIS
LIN {X -0.186,Y -650.573,Z 1375.429,A 0.000,B 0.000,C 90.000,E1 113.259} C_DIS
LIN {X -0.095,Y -648.639,Z 1375.428,A 0.000,B 0.000,C 90.000,E1 113.131} C_DIS
LIN {X 0.307,Y -641.487,Z 1375.427,A 0.000,B 0.000,C 90.000,E1 112.770} C_DIS
LIN {X 0.252,Y -637.778,Z 1375.426,A 0.000,B 0.000,C 90.000,E1 112.642} C_DIS
LIN {X -0.126,Y -622.426,Z 1375.424,A 0.000,B 0.000,C 90.000,E1 112.259} C_DIS
LIN {X -0.159,Y -622.351,Z 1375.424,A 0.000,B 0.000,C 90.000,E1 112.259} C_DIS
LIN {X 0.013,Y -632.319,Z 1375.418,A 0.000,B 0.000,C 90.000,E1 111.173} C_DIS
LIN {X -0.140,Y -637.713,Z 1375.414,A 0.000,B 0.000,C 90.000,E1 110.556} C_DIS
LIN {X -0.265,Y -642.353,Z 1375.411,A 0.000,B 0.000,C 90.000,E1 109.939} C_DIS
LIN {X 0.252,Y -646.324,Z 1375.407,A 0.000,B 0.000,C 90.000,E1 109.268} C_DIS
LIN {X 0.088,Y -651.034,Z 1375.402,A 0.000,B 0.000,C 90.000,E1 108.417} C_DIS
LIN {X -0.109,Y -654.750,Z 1375.398,A 0.000,B 0.000,C 90.000,E1 107.692} C_DIS
LIN {X -0.353,Y -657.093,Z 1375.396,A 0.000,B 0.000,C 90.000,E1 107.221} C_DIS
LIN {X 0.239,Y -659.130,Z 1375.393,A 0.000,B 0.000,C 90.000,E1 106.677} C_DIS
LIN {X 0.132,Y -660.099,Z 1375.391,A 0.000,B 0.000,C 90.000,E1 106.441} C_DIS
LIN {X 0.010,Y -662.454,Z 1375.387,A 0.000,B 0.000,C 90.000,E1 105.717} C_DIS
LIN {X -0.270,Y -664.148,Z 1375.383,A 0.000,B 0.000,C 90.000,E1 105.009} C_DIS
LIN {X 0.198,Y -665.080,Z 1375.381,A 0.000,B 0.000,C 90.000,E1 104.481} C_DIS
LIN {X -0.051,Y -666.030,Z 1375.377,A 0.000,B 0.000,C 90.000,E1 103.772} C_DIS
LIN {X -0.213,Y -666.470,Z 1375.374,A 0.000,B 0.000,C 90.000,E1 103.300} C_DIS
LIN {X 0.278,Y -666.659,Z 1375.371,A 0.000,B 0.000,C 90.000,E1 102.771} C_DIS
LIN {X 0.038,Y -666.579,Z 1375.367,A 0.000,B 0.000,C 90.000,E1 102.063} C_DIS
LIN {X -0.124,Y -666.324,Z 1375.364,A 0.000,B 0.000,C 90.000,E1 101.591} C_DIS
LIN {X 0.233,Y -665.812,Z 1375.362,A 0.000,B 0.000,C 90.000,E1 101.074} C_DIS
LIN {X -0.025,Y -664.642,Z 1375.358,A 0.000,B 0.000,C 90.000,E1 100.366} C_DIS
LIN {X -0.323,Y -663.631,Z 1375.355,A 0.000,B 0.000,C 90.000,E1 99.905} C_DIS
LIN {X 0.140,Y -662.424,Z 1375.352,A 0.000,B 0.000,C 90.000,E1 99.378} C_DIS
LIN {X -0.168,Y -660.976,Z 1375.349,A 0.000,B 0.000,C 90.000,E1 98.916} C_DIS
LIN {X 0.059,Y -658.384,Z 1375.345,A 0.000,B 0.000,C 90.000,E1 98.163} C_DIS
LIN {X -0.268,Y -656.429,Z 1375.343,A 0.000,B 0.000,C 90.000,E1 97.701} C_DIS
LIN {X 0.044,Y -654.284,Z 1375.340,A 0.000,B 0.000,C 90.000,E1 97.182} C_DIS
LIN {X -0.305,Y -651.862,Z 1375.337,A 0.000,B 0.000,C 90.000,E1 96.720} C_DIS
LIN {X -0.136,Y -648.513,Z 1375.334,A 0.000,B 0.000,C 90.000,E1 96.087} C_DIS
LIN {X -0.170,Y -643.304,Z 1375.329,A 0.000,B 0.000,C 90.000,E1 95.220} C_DIS
LIN {X -0.077,Y -639.408,Z 1375.325,A 0.000,B 0.000,C 90.000,E1 94.588} C_DIS
LIN {X -0.020,Y -635.049,Z 1375.322,A 0.000,B 0.000,C 90.000,E1 93.955} C_DIS
LIN {X 0.092,Y -631.153,Z 1375.319,A 0.000,B 0.000,C 90.000,E1 93.440} C_DIS
LIN {X 0.075,Y -625.407,Z 1375.316,A 0.000,B 0.000,C 90.000,E1 92.808} C_DIS
LIN {X 0.205,Y -617.929,Z 1375.312,A 0.000,B 0.000,C 90.000,E1 92.064} C_DIS
LIN {X -0.158,Y -610.075,Z 1375.308,A 0.000,B 0.000,C 90.000,E1 91.375} C_DIS
LIN {X -0.246,Y -605.816,Z 1375.306,A 0.000,B 0.000,C 90.000,E1 91.031} C_DIS
LIN {X -0.182,Y -602.924,Z 1375.304,A 0.000,B 0.000,C 90.000,E1 90.802} C_DIS
LIN {X 0.231,Y -596.459,Z 1375.302,A 0.000,B 0.000,C 90.000,E1 90.344} C_DIS
LIN {X 0.082,Y -589.598,Z 1375.300,A 0.000,B 0.000,C 90.000,E1 90.000} C_DIS
LIN {X 0.225,Y -579.817,Z 1375.298,A 0.000,B 0.000,C 90.000,E1 89.542} C_DIS
LIN {X -0.158,Y -576.978,Z 1375.297,A 0.000,B 0.000,C 90.000,E1 89.427} C_DIS
LIN {X -0.164,Y -574.134,Z 1375.295,A 0.000,B 0.000,C 90.000,E1 89.141} C_DIS
LIN {X -0.205,Y -574.103,Z 1375.295,A 0.000,B 0.000,C 90.000,E1 89.141} C_DIS
LIN {X 0.088,Y -573.585,Z 1375.293,A 0.000,B 0.000,C 90.000,E1 88.797} C_DIS
LIN {X 0.176,Y -573.922,Z 1375.290,A 0.000,B 0.000,C 90.000,E1 88.108} C_DIS
LIN {X 0.206,Y -575.753,Z 1375.278,A 0.000,B 0.000,C 90.000,E1 85.931} C_DIS
LIN {X -0.030,Y -578.279,Z 1375.264,A 0.000,B 0.000,C 90.000,E1 83.514} C_DIS
LIN {X -0.266,Y -579.870,Z 1375.256,A 0.000,B 0.000,C 90.000,E1 82.186} C_DIS
LIN {X -0.157,Y -581.824,Z 1375.248,A 0.000,B 0.000,C 90.000,E1 80.557} C_DIS
LIN {X -0.235,Y -583.378,Z 1375.240,A 0.000,B 0.000,C 90.000,E1 79.218} C_DIS
LIN {X -0.297,Y -584.743,Z 1375.233,A 0.000,B 0.000,C 90.000,E1 77.881} C_DIS
LIN {X -0.089,Y -585.930,Z 1375.225,A 0.000,B 0.000,C 90.000,E1 76.520} C_DIS
LIN {X 0.004,Y -586.941,Z 1375.218,A 0.000,B 0.000,C 90.000,E1 75.172} C_DIS
LIN {X -0.151,Y -587.865,Z 1375.210,A 0.000,B 0.000,C 90.000,E1 73.850} C_DIS
LIN {X -0.034,Y -588.843,Z 1375.201,A 0.000,B 0.000,C 90.000,E1 72.236} C_DIS
LIN {X 0.173,Y -589.431,Z 1375.195,A 0.000,B 0.000,C 90.000,E1 71.148} C_DIS
LIN {X -0.062,Y -590.362,Z 1375.187,A 0.000,B 0.000,C 90.000,E1 69.571} C_DIS
LIN {X 0.253,Y -591.609,Z 1375.175,A 0.000,B 0.000,C 90.000,E1 67.411} C_DIS
LIN {X -0.052,Y -592.802,Z 1375.166,A 0.000,B 0.000,C 90.000,E1 65.845} C_DIS
LIN {X -0.244,Y -593.949,Z 1375.158,A 0.000,B 0.000,C 90.000,E1 64.537} C_DIS
LIN {X 0.004,Y -595.170,Z 1375.150,A 0.000,B 0.000,C 90.000,E1 62.922} C_DIS
LIN {X 0.113,Y -596.876,Z 1375.138,A 0.000,B 0.000,C 90.000,E1 60.795} C_DIS
LIN {X -0.026,Y -598.121,Z 1375.130,A 0.000,B 0.000,C 90.000,E1 59.488} C_DIS
